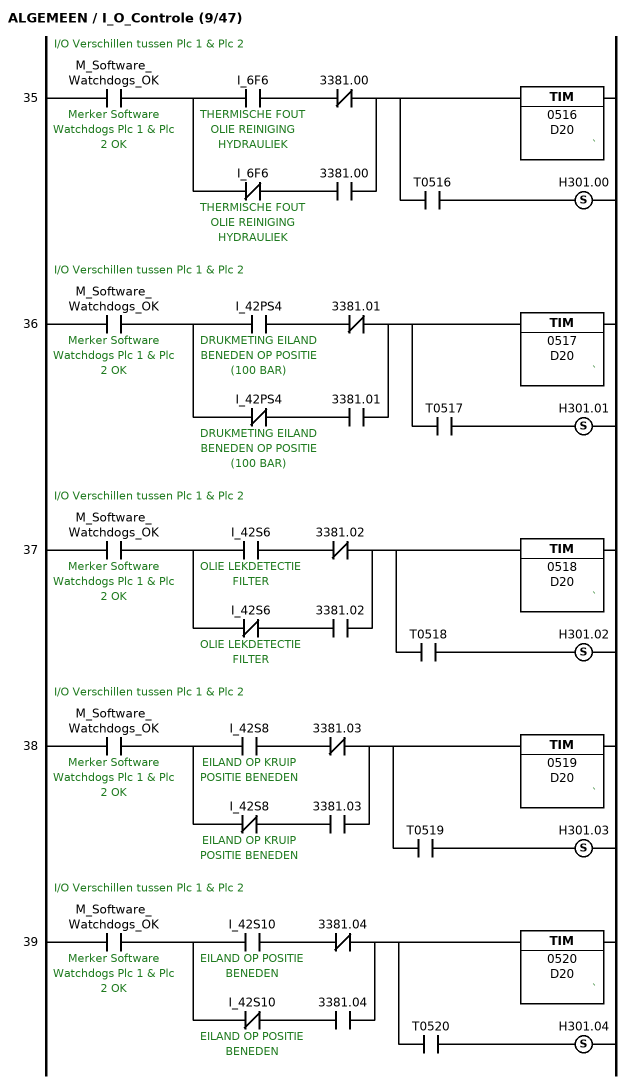
; [picture p24: ALGEMEEN / I_O_Controle, rungs 35-39]
; rung 35: I/O Verschillen tussen Plc 1 & Plc 2
LD M_Software_Watchdogs_OK  ; Merker Software Watchdogs Plc 1 & Plc 2 OK
LD I_6F6  ; THERMISCHE FOUT OLIE REINIGING HYDRAULIEK
ANDNOT 3381.00
LDNOT I_6F6  ; THERMISCHE FOUT OLIE REINIGING HYDRAULIEK
AND 3381.00
ORLD
ANDLD
TIM 0516 D20  ; `
AND T0516
SET H301.00
; rung 36: I/O Verschillen tussen Plc 1 & Plc 2
LD M_Software_Watchdogs_OK  ; Merker Software Watchdogs Plc 1 & Plc 2 OK
LD I_42PS4  ; DRUKMETING EILAND BENEDEN OP POSITIE (100 BAR)
ANDNOT 3381.01
LDNOT I_42PS4  ; DRUKMETING EILAND BENEDEN OP POSITIE (100 BAR)
AND 3381.01
ORLD
ANDLD
TIM 0517 D20  ; `
AND T0517
SET H301.01
; rung 37: I/O Verschillen tussen Plc 1 & Plc 2
LD M_Software_Watchdogs_OK  ; Merker Software Watchdogs Plc 1 & Plc 2 OK
LD I_42S6  ; OLIE LEKDETECTIE FILTER
ANDNOT 3381.02
LDNOT I_42S6  ; OLIE LEKDETECTIE FILTER
AND 3381.02
ORLD
ANDLD
TIM 0518 D20  ; `
AND T0518
SET H301.02
; rung 38: I/O Verschillen tussen Plc 1 & Plc 2
LD M_Software_Watchdogs_OK  ; Merker Software Watchdogs Plc 1 & Plc 2 OK
LD I_42S8  ; EILAND OP KRUIP POSITIE BENEDEN
ANDNOT 3381.03
LDNOT I_42S8  ; EILAND OP KRUIP POSITIE BENEDEN
AND 3381.03
ORLD
ANDLD
TIM 0519 D20  ; `
AND T0519
SET H301.03
; rung 39: I/O Verschillen tussen Plc 1 & Plc 2
LD M_Software_Watchdogs_OK  ; Merker Software Watchdogs Plc 1 & Plc 2 OK
LD I_42S10  ; EILAND OP POSITIE BENEDEN
ANDNOT 3381.04
LDNOT I_42S10  ; EILAND OP POSITIE BENEDEN
AND 3381.04
ORLD
ANDLD
TIM 0520 D20  ; `
AND T0520
SET H301.04

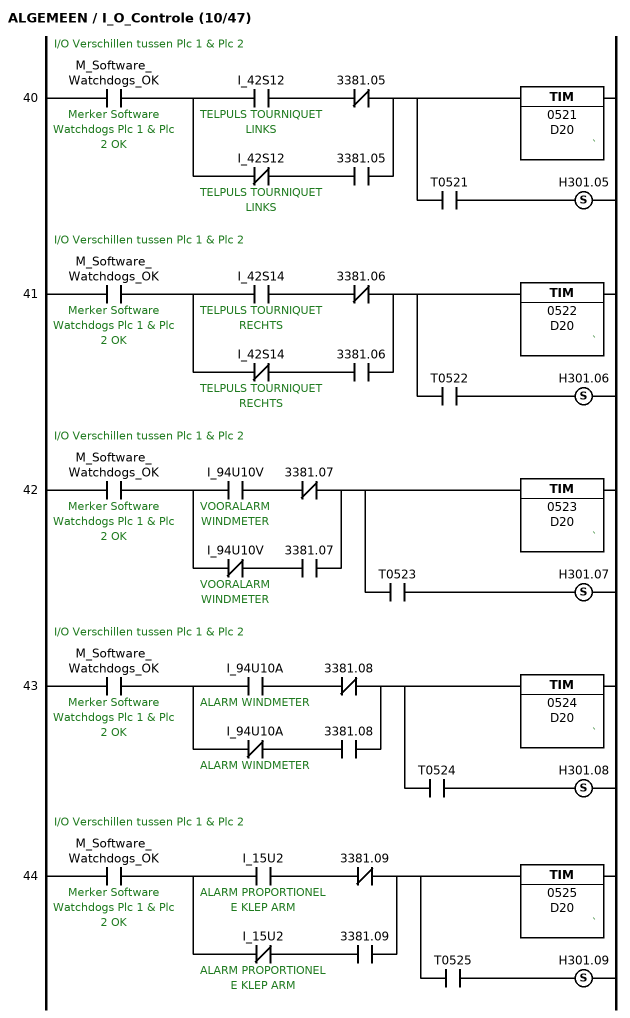
; rung 40: I/O Verschillen tussen Plc 1 & Plc 2
LD M_Software_Watchdogs_OK  ; Merker Software Watchdogs Plc 1 & Plc 2 OK
LD I_42S12  ; TELPULS TOURNIQUET LINKS
ANDNOT 3381.05
LDNOT I_42S12  ; TELPULS TOURNIQUET LINKS
AND 3381.05
ORLD
ANDLD
TIM 0521 D20  ; `
AND T0521
SET H301.05
; rung 41: I/O Verschillen tussen Plc 1 & Plc 2
LD M_Software_Watchdogs_OK  ; Merker Software Watchdogs Plc 1 & Plc 2 OK
LD I_42S14  ; TELPULS TOURNIQUET RECHTS
ANDNOT 3381.06
LDNOT I_42S14  ; TELPULS TOURNIQUET RECHTS
AND 3381.06
ORLD
ANDLD
TIM 0522 D20  ; `
AND T0522
SET H301.06
; rung 42: I/O Verschillen tussen Plc 1 & Plc 2
LD M_Software_Watchdogs_OK  ; Merker Software Watchdogs Plc 1 & Plc 2 OK
LD I_94U10V  ; VOORALARM WINDMETER
ANDNOT 3381.07
LDNOT I_94U10V  ; VOORALARM WINDMETER
AND 3381.07
ORLD
ANDLD
TIM 0523 D20  ; `
AND T0523
SET H301.07
; rung 43: I/O Verschillen tussen Plc 1 & Plc 2
LD M_Software_Watchdogs_OK  ; Merker Software Watchdogs Plc 1 & Plc 2 OK
LD I_94U10A  ; ALARM WINDMETER
ANDNOT 3381.08
LDNOT I_94U10A  ; ALARM WINDMETER
AND 3381.08
ORLD
ANDLD
TIM 0524 D20  ; `
AND T0524
SET H301.08
; rung 44: I/O Verschillen tussen Plc 1 & Plc 2
LD M_Software_Watchdogs_OK  ; Merker Software Watchdogs Plc 1 & Plc 2 OK
LD I_15U2  ; ALARM PROPORTIONELE KLEP ARM
ANDNOT 3381.09
LDNOT I_15U2  ; ALARM PROPORTIONELE KLEP ARM
AND 3381.09
ORLD
ANDLD
TIM 0525 D20  ; `
AND T0525
SET H301.09

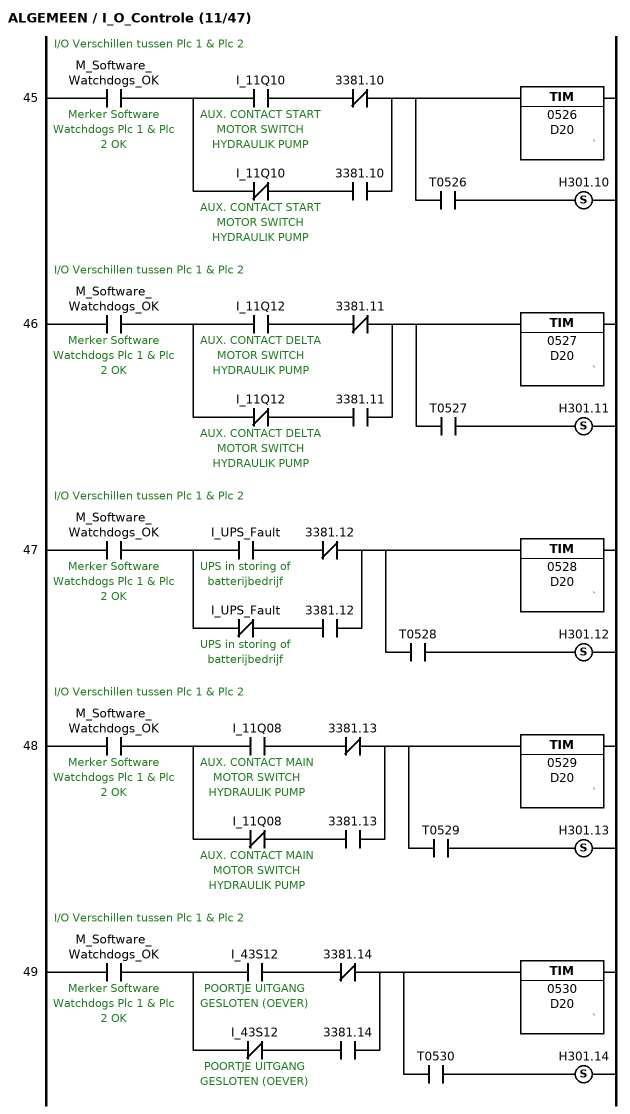
; rung 45: I/O Verschillen tussen Plc 1 & Plc 2
LD M_Software_Watchdogs_OK  ; Merker Software Watchdogs Plc 1 & Plc 2 OK
LD I_11Q10  ; AUX. CONTACT START MOTOR SWITCH HYDRAULIK PUMP
ANDNOT 3381.10
LDNOT I_11Q10  ; AUX. CONTACT START MOTOR SWITCH HYDRAULIK PUMP
AND 3381.10
ORLD
ANDLD
TIM 0526 D20  ; `
AND T0526
SET H301.10
; rung 46: I/O Verschillen tussen Plc 1 & Plc 2
LD M_Software_Watchdogs_OK  ; Merker Software Watchdogs Plc 1 & Plc 2 OK
LD I_11Q12  ; AUX. CONTACT DELTA MOTOR SWITCH HYDRAULIK PUMP
ANDNOT 3381.11
LDNOT I_11Q12  ; AUX. CONTACT DELTA MOTOR SWITCH HYDRAULIK PUMP
AND 3381.11
ORLD
ANDLD
TIM 0527 D20  ; `
AND T0527
SET H301.11
; rung 47: I/O Verschillen tussen Plc 1 & Plc 2
LD M_Software_Watchdogs_OK  ; Merker Software Watchdogs Plc 1 & Plc 2 OK
LD I_UPS_Fault  ; UPS in storing of batterijbedrijf
ANDNOT 3381.12
LDNOT I_UPS_Fault  ; UPS in storing of batterijbedrijf
AND 3381.12
ORLD
ANDLD
TIM 0528 D20  ; `
AND T0528
SET H301.12
; rung 48: I/O Verschillen tussen Plc 1 & Plc 2
LD M_Software_Watchdogs_OK  ; Merker Software Watchdogs Plc 1 & Plc 2 OK
LD I_11Q08  ; AUX. CONTACT MAIN MOTOR SWITCH HYDRAULIK PUMP
ANDNOT 3381.13
LDNOT I_11Q08  ; AUX. CONTACT MAIN MOTOR SWITCH HYDRAULIK PUMP
AND 3381.13
ORLD
ANDLD
TIM 0529 D20  ; `
AND T0529
SET H301.13
; rung 49: I/O Verschillen tussen Plc 1 & Plc 2
LD M_Software_Watchdogs_OK  ; Merker Software Watchdogs Plc 1 & Plc 2 OK
LD I_43S12  ; POORTJE UITGANG GESLOTEN (OEVER)
ANDNOT 3381.14
LDNOT I_43S12  ; POORTJE UITGANG GESLOTEN (OEVER)
AND 3381.14
ORLD
ANDLD
TIM 0530 D20  ; `
AND T0530
SET H301.14

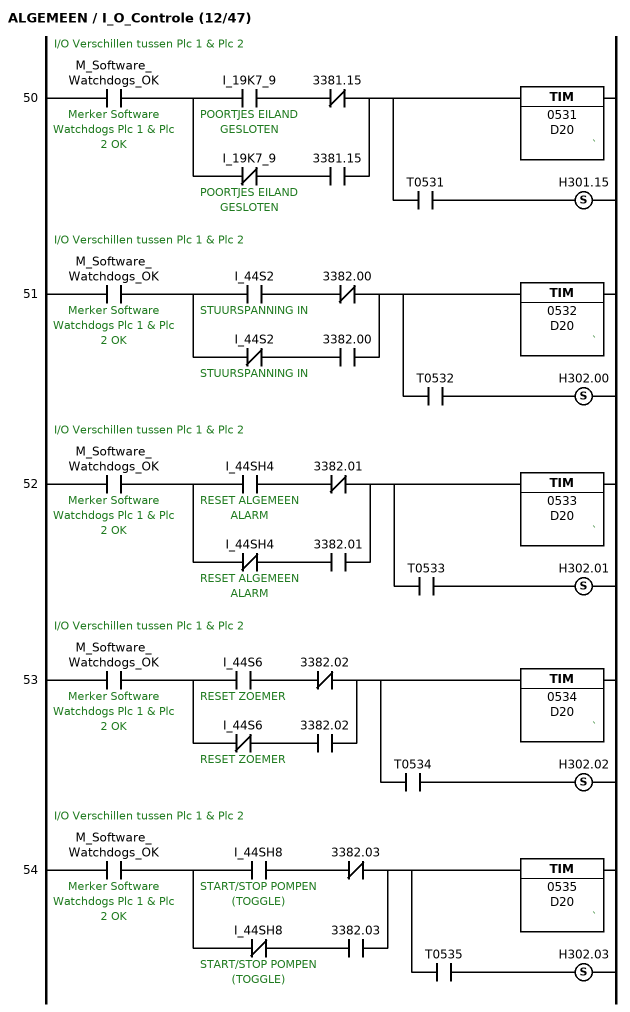
; rung 50: I/O Verschillen tussen Plc 1 & Plc 2
LD M_Software_Watchdogs_OK  ; Merker Software Watchdogs Plc 1 & Plc 2 OK
LD I_19K7_9  ; POORTJES EILAND GESLOTEN
ANDNOT 3381.15
LDNOT I_19K7_9  ; POORTJES EILAND GESLOTEN
AND 3381.15
ORLD
ANDLD
TIM 0531 D20  ; `
AND T0531
SET H301.15
; rung 51: I/O Verschillen tussen Plc 1 & Plc 2
LD M_Software_Watchdogs_OK  ; Merker Software Watchdogs Plc 1 & Plc 2 OK
LD I_44S2  ; STUURSPANNING IN
ANDNOT 3382.00
LDNOT I_44S2  ; STUURSPANNING IN
AND 3382.00
ORLD
ANDLD
TIM 0532 D20  ; `
AND T0532
SET H302.00
; rung 52: I/O Verschillen tussen Plc 1 & Plc 2
LD M_Software_Watchdogs_OK  ; Merker Software Watchdogs Plc 1 & Plc 2 OK
LD I_44SH4  ; RESET ALGEMEEN ALARM
ANDNOT 3382.01
LDNOT I_44SH4  ; RESET ALGEMEEN ALARM
AND 3382.01
ORLD
ANDLD
TIM 0533 D20  ; `
AND T0533
SET H302.01
; rung 53: I/O Verschillen tussen Plc 1 & Plc 2
LD M_Software_Watchdogs_OK  ; Merker Software Watchdogs Plc 1 & Plc 2 OK
LD I_44S6  ; RESET ZOEMER
ANDNOT 3382.02
LDNOT I_44S6  ; RESET ZOEMER
AND 3382.02
ORLD
ANDLD
TIM 0534 D20  ; `
AND T0534
SET H302.02
; rung 54: I/O Verschillen tussen Plc 1 & Plc 2
LD M_Software_Watchdogs_OK  ; Merker Software Watchdogs Plc 1 & Plc 2 OK
LD I_44SH8  ; START/STOP POMPEN (TOGGLE)
ANDNOT 3382.03
LDNOT I_44SH8  ; START/STOP POMPEN (TOGGLE)
AND 3382.03
ORLD
ANDLD
TIM 0535 D20  ; `
AND T0535
SET H302.03

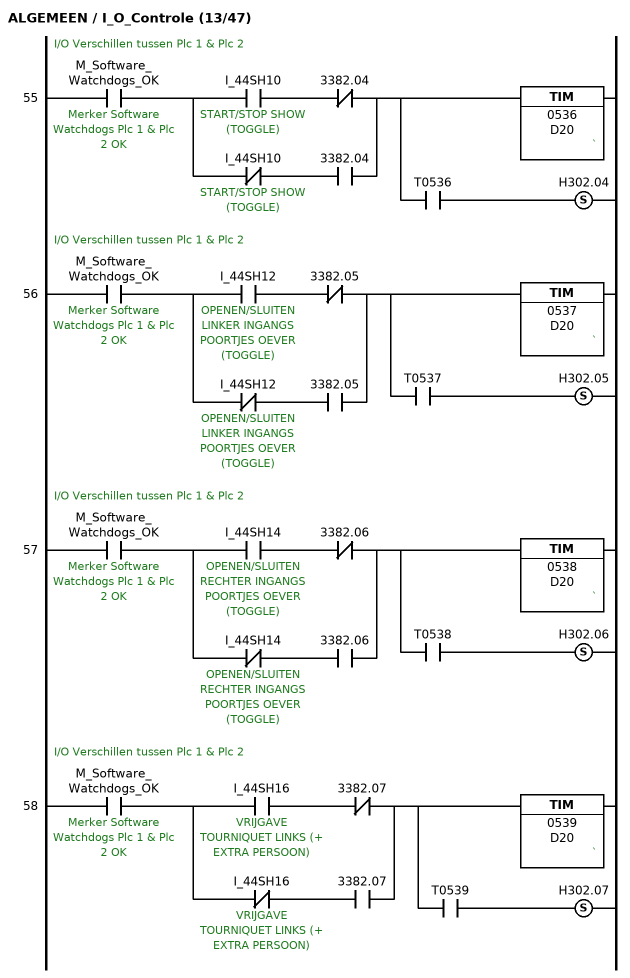
; rung 55: I/O Verschillen tussen Plc 1 & Plc 2
LD M_Software_Watchdogs_OK  ; Merker Software Watchdogs Plc 1 & Plc 2 OK
LD I_44SH10  ; START/STOP SHOW (TOGGLE)
ANDNOT 3382.04
LDNOT I_44SH10  ; START/STOP SHOW (TOGGLE)
AND 3382.04
ORLD
ANDLD
TIM 0536 D20  ; `
AND T0536
SET H302.04
; rung 56: I/O Verschillen tussen Plc 1 & Plc 2
LD M_Software_Watchdogs_OK  ; Merker Software Watchdogs Plc 1 & Plc 2 OK
LD I_44SH12  ; OPENEN/SLUITEN LINKER INGANGS POORTJES OEVER  (TOGGLE)
ANDNOT 3382.05
LDNOT I_44SH12  ; OPENEN/SLUITEN LINKER INGANGS POORTJES OEVER  (TOGGLE)
AND 3382.05
ORLD
ANDLD
TIM 0537 D20  ; `
AND T0537
SET H302.05
; rung 57: I/O Verschillen tussen Plc 1 & Plc 2
LD M_Software_Watchdogs_OK  ; Merker Software Watchdogs Plc 1 & Plc 2 OK
LD I_44SH14  ; OPENEN/SLUITEN RECHTER INGANGS POORTJES OEVER  (TOGGLE)
ANDNOT 3382.06
LDNOT I_44SH14  ; OPENEN/SLUITEN RECHTER INGANGS POORTJES OEVER  (TOGGLE)
AND 3382.06
ORLD
ANDLD
TIM 0538 D20  ; `
AND T0538
SET H302.06
; rung 58: I/O Verschillen tussen Plc 1 & Plc 2
LD M_Software_Watchdogs_OK  ; Merker Software Watchdogs Plc 1 & Plc 2 OK
LD I_44SH16  ; VRIJGAVE TOURNIQUET LINKS (+ EXTRA PERSOON)
ANDNOT 3382.07
LDNOT I_44SH16  ; VRIJGAVE TOURNIQUET LINKS (+ EXTRA PERSOON)
AND 3382.07
ORLD
ANDLD
TIM 0539 D20  ; `
AND T0539
SET H302.07

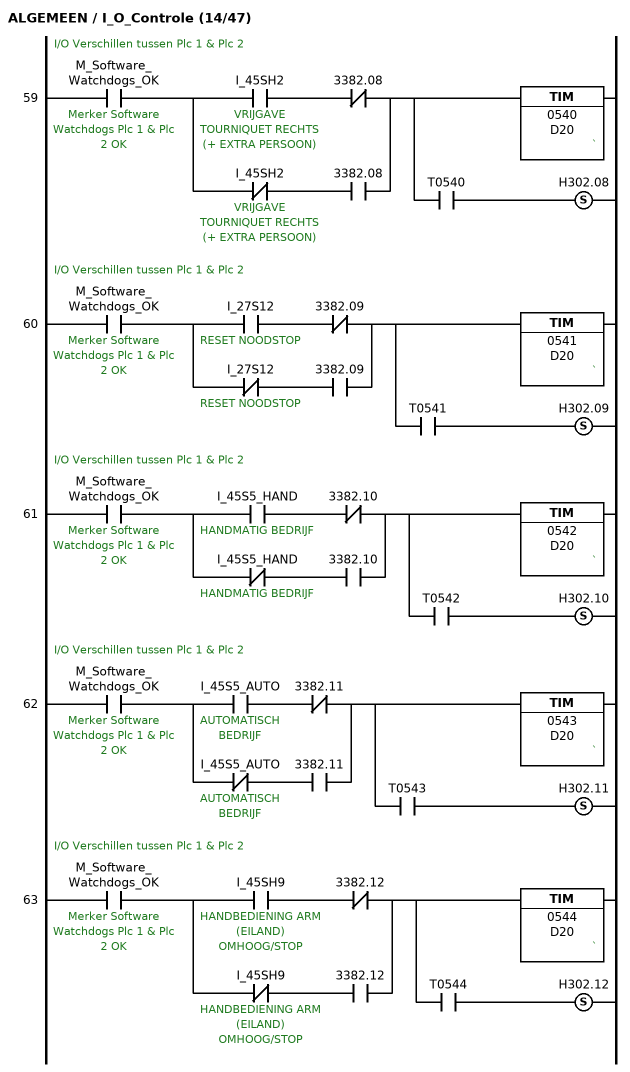
; rung 59: I/O Verschillen tussen Plc 1 & Plc 2
LD M_Software_Watchdogs_OK  ; Merker Software Watchdogs Plc 1 & Plc 2 OK
LD I_45SH2  ; VRIJGAVE TOURNIQUET RECHTS (+ EXTRA PERSOON)
ANDNOT 3382.08
LDNOT I_45SH2  ; VRIJGAVE TOURNIQUET RECHTS (+ EXTRA PERSOON)
AND 3382.08
ORLD
ANDLD
TIM 0540 D20  ; `
AND T0540
SET H302.08
; rung 60: I/O Verschillen tussen Plc 1 & Plc 2
LD M_Software_Watchdogs_OK  ; Merker Software Watchdogs Plc 1 & Plc 2 OK
LD I_27S12  ; RESET NOODSTOP
ANDNOT 3382.09
LDNOT I_27S12  ; RESET NOODSTOP
AND 3382.09
ORLD
ANDLD
TIM 0541 D20  ; `
AND T0541
SET H302.09
; rung 61: I/O Verschillen tussen Plc 1 & Plc 2
LD M_Software_Watchdogs_OK  ; Merker Software Watchdogs Plc 1 & Plc 2 OK
LD I_45S5_HAND  ; HANDMATIG BEDRIJF
ANDNOT 3382.10
LDNOT I_45S5_HAND  ; HANDMATIG BEDRIJF
AND 3382.10
ORLD
ANDLD
TIM 0542 D20  ; `
AND T0542
SET H302.10
; rung 62: I/O Verschillen tussen Plc 1 & Plc 2
LD M_Software_Watchdogs_OK  ; Merker Software Watchdogs Plc 1 & Plc 2 OK
LD I_45S5_AUTO  ; AUTOMATISCH BEDRIJF
ANDNOT 3382.11
LDNOT I_45S5_AUTO  ; AUTOMATISCH BEDRIJF
AND 3382.11
ORLD
ANDLD
TIM 0543 D20  ; `
AND T0543
SET H302.11
; rung 63: I/O Verschillen tussen Plc 1 & Plc 2
LD M_Software_Watchdogs_OK  ; Merker Software Watchdogs Plc 1 & Plc 2 OK
LD I_45SH9  ; HANDBEDIENING ARM (EILAND) OMHOOG/STOP
ANDNOT 3382.12
LDNOT I_45SH9  ; HANDBEDIENING ARM (EILAND) OMHOOG/STOP
AND 3382.12
ORLD
ANDLD
TIM 0544 D20  ; `
AND T0544
SET H302.12

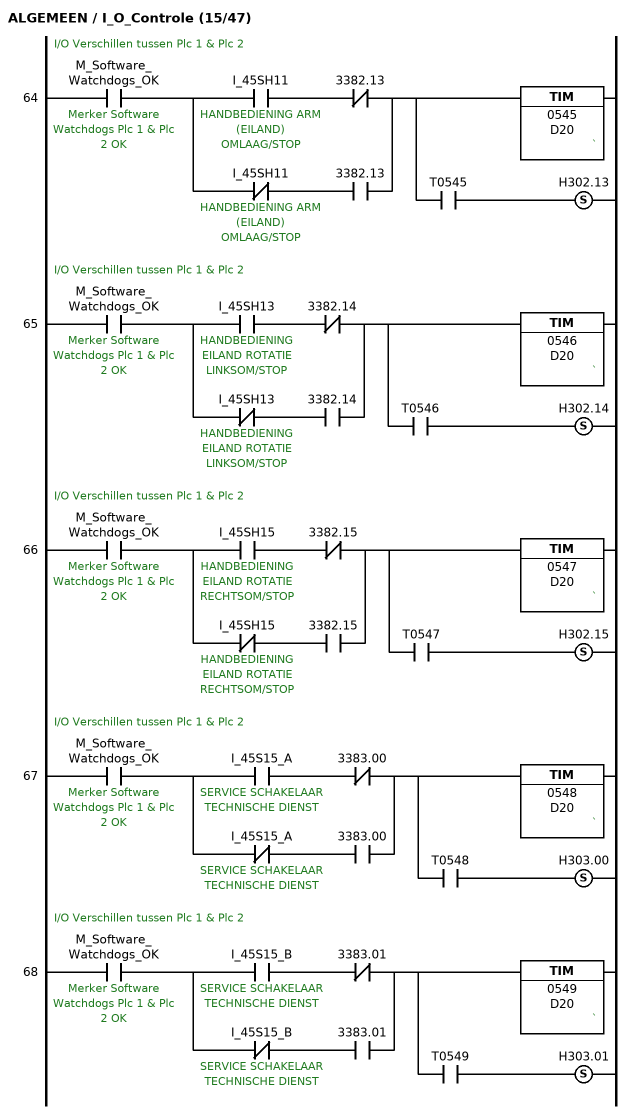
; rung 64: I/O Verschillen tussen Plc 1 & Plc 2
LD M_Software_Watchdogs_OK  ; Merker Software Watchdogs Plc 1 & Plc 2 OK
LD I_45SH11  ; HANDBEDIENING ARM (EILAND) OMLAAG/STOP
ANDNOT 3382.13
LDNOT I_45SH11  ; HANDBEDIENING ARM (EILAND) OMLAAG/STOP
AND 3382.13
ORLD
ANDLD
TIM 0545 D20  ; `
AND T0545
SET H302.13
; rung 65: I/O Verschillen tussen Plc 1 & Plc 2
LD M_Software_Watchdogs_OK  ; Merker Software Watchdogs Plc 1 & Plc 2 OK
LD I_45SH13  ; HANDBEDIENING EILAND ROTATIE LINKSOM/STOP
ANDNOT 3382.14
LDNOT I_45SH13  ; HANDBEDIENING EILAND ROTATIE LINKSOM/STOP
AND 3382.14
ORLD
ANDLD
TIM 0546 D20  ; `
AND T0546
SET H302.14
; rung 66: I/O Verschillen tussen Plc 1 & Plc 2
LD M_Software_Watchdogs_OK  ; Merker Software Watchdogs Plc 1 & Plc 2 OK
LD I_45SH15  ; HANDBEDIENING EILAND ROTATIE RECHTSOM/STOP
ANDNOT 3382.15
LDNOT I_45SH15  ; HANDBEDIENING EILAND ROTATIE RECHTSOM/STOP
AND 3382.15
ORLD
ANDLD
TIM 0547 D20  ; `
AND T0547
SET H302.15
; rung 67: I/O Verschillen tussen Plc 1 & Plc 2
LD M_Software_Watchdogs_OK  ; Merker Software Watchdogs Plc 1 & Plc 2 OK
LD I_45S15_A  ; SERVICE SCHAKELAAR TECHNISCHE DIENST
ANDNOT 3383.00
LDNOT I_45S15_A  ; SERVICE SCHAKELAAR TECHNISCHE DIENST
AND 3383.00
ORLD
ANDLD
TIM 0548 D20  ; `
AND T0548
SET H303.00
; rung 68: I/O Verschillen tussen Plc 1 & Plc 2
LD M_Software_Watchdogs_OK  ; Merker Software Watchdogs Plc 1 & Plc 2 OK
LD I_45S15_B  ; SERVICE SCHAKELAAR TECHNISCHE DIENST
ANDNOT 3383.01
LDNOT I_45S15_B  ; SERVICE SCHAKELAAR TECHNISCHE DIENST
AND 3383.01
ORLD
ANDLD
TIM 0549 D20  ; `
AND T0549
SET H303.01

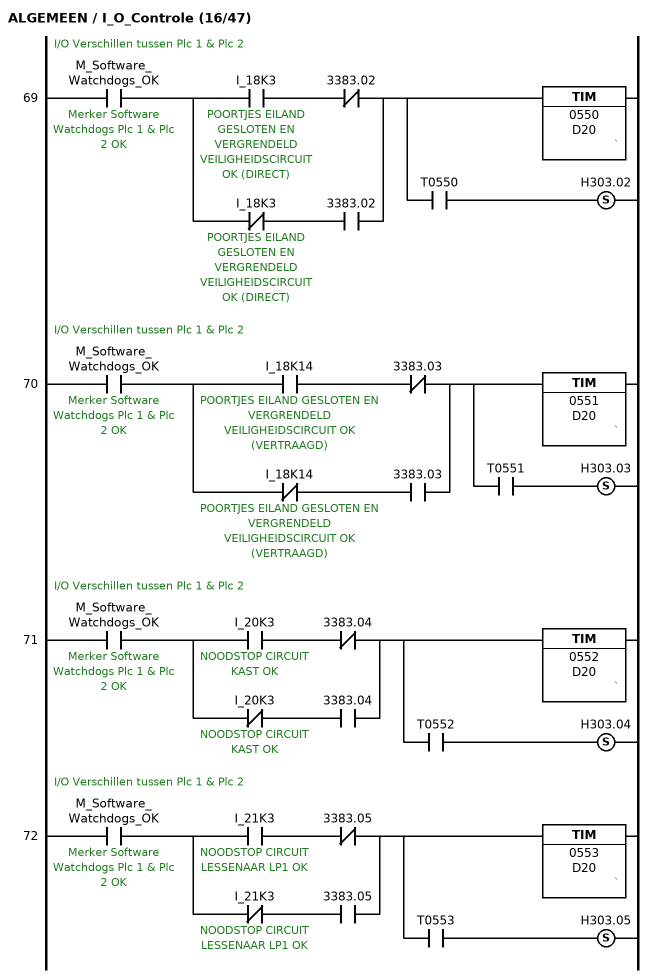
; rung 69: I/O Verschillen tussen Plc 1 & Plc 2
LD M_Software_Watchdogs_OK  ; Merker Software Watchdogs Plc 1 & Plc 2 OK
LD I_18K3  ; POORTJES EILAND GESLOTEN EN VERGRENDELD VEILIGHEIDSCIRCUIT OK (DIRECT)
ANDNOT 3383.02
LDNOT I_18K3  ; POORTJES EILAND GESLOTEN EN VERGRENDELD VEILIGHEIDSCIRCUIT OK (DIRECT)
AND 3383.02
ORLD
ANDLD
TIM 0550 D20  ; `
AND T0550
SET H303.02
; rung 70: I/O Verschillen tussen Plc 1 & Plc 2
LD M_Software_Watchdogs_OK  ; Merker Software Watchdogs Plc 1 & Plc 2 OK
LD I_18K14  ; POORTJES EILAND GESLOTEN EN VERGRENDELD VEILIGHEIDSCIRCUIT OK (VERTRAAGD)
ANDNOT 3383.03
LDNOT I_18K14  ; POORTJES EILAND GESLOTEN EN VERGRENDELD VEILIGHEIDSCIRCUIT OK (VERTRAAGD)
AND 3383.03
ORLD
ANDLD
TIM 0551 D20  ; `
AND T0551
SET H303.03
; rung 71: I/O Verschillen tussen Plc 1 & Plc 2
LD M_Software_Watchdogs_OK  ; Merker Software Watchdogs Plc 1 & Plc 2 OK
LD I_20K3  ; NOODSTOP CIRCUIT KAST OK
ANDNOT 3383.04
LDNOT I_20K3  ; NOODSTOP CIRCUIT KAST OK
AND 3383.04
ORLD
ANDLD
TIM 0552 D20  ; `
AND T0552
SET H303.04
; rung 72: I/O Verschillen tussen Plc 1 & Plc 2
LD M_Software_Watchdogs_OK  ; Merker Software Watchdogs Plc 1 & Plc 2 OK
LD I_21K3  ; NOODSTOP CIRCUIT LESSENAAR LP1 OK
ANDNOT 3383.05
LDNOT I_21K3  ; NOODSTOP CIRCUIT LESSENAAR LP1 OK
AND 3383.05
ORLD
ANDLD
TIM 0553 D20  ; `
AND T0553
SET H303.05

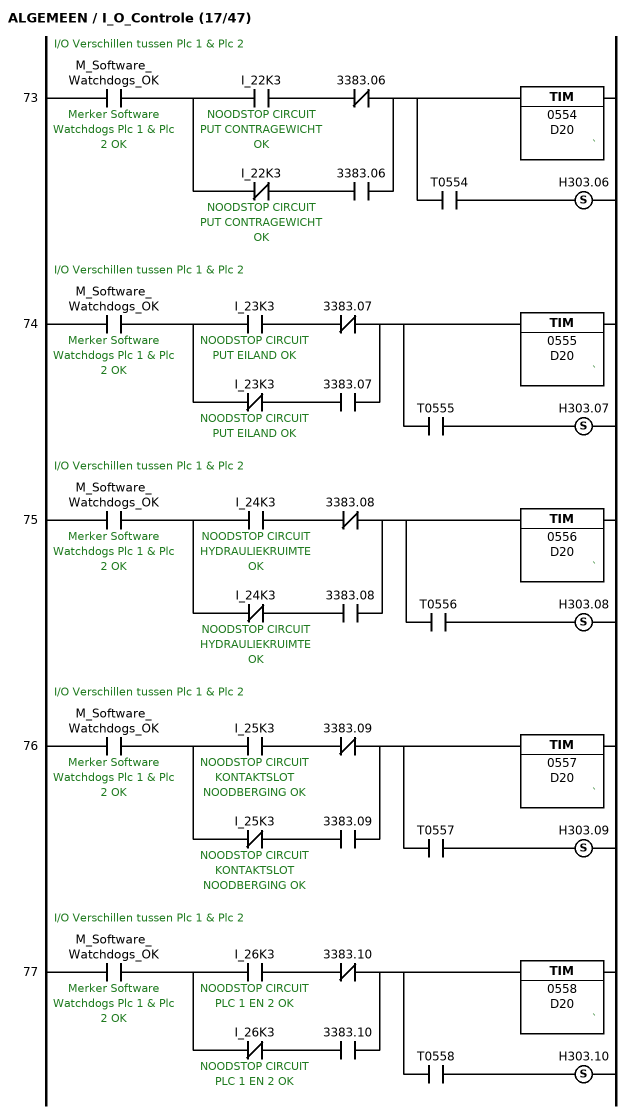
; rung 73: I/O Verschillen tussen Plc 1 & Plc 2
LD M_Software_Watchdogs_OK  ; Merker Software Watchdogs Plc 1 & Plc 2 OK
LD I_22K3  ; NOODSTOP CIRCUIT PUT CONTRAGEWICHT OK
ANDNOT 3383.06
LDNOT I_22K3  ; NOODSTOP CIRCUIT PUT CONTRAGEWICHT OK
AND 3383.06
ORLD
ANDLD
TIM 0554 D20  ; `
AND T0554
SET H303.06
; rung 74: I/O Verschillen tussen Plc 1 & Plc 2
LD M_Software_Watchdogs_OK  ; Merker Software Watchdogs Plc 1 & Plc 2 OK
LD I_23K3  ; NOODSTOP CIRCUIT PUT EILAND OK
ANDNOT 3383.07
LDNOT I_23K3  ; NOODSTOP CIRCUIT PUT EILAND OK
AND 3383.07
ORLD
ANDLD
TIM 0555 D20  ; `
AND T0555
SET H303.07
; rung 75: I/O Verschillen tussen Plc 1 & Plc 2
LD M_Software_Watchdogs_OK  ; Merker Software Watchdogs Plc 1 & Plc 2 OK
LD I_24K3  ; NOODSTOP CIRCUIT HYDRAULIEKRUIMTE OK
ANDNOT 3383.08
LDNOT I_24K3  ; NOODSTOP CIRCUIT HYDRAULIEKRUIMTE OK
AND 3383.08
ORLD
ANDLD
TIM 0556 D20  ; `
AND T0556
SET H303.08
; rung 76: I/O Verschillen tussen Plc 1 & Plc 2
LD M_Software_Watchdogs_OK  ; Merker Software Watchdogs Plc 1 & Plc 2 OK
LD I_25K3  ; NOODSTOP CIRCUIT KONTAKTSLOT NOODBERGING OK
ANDNOT 3383.09
LDNOT I_25K3  ; NOODSTOP CIRCUIT KONTAKTSLOT NOODBERGING OK
AND 3383.09
ORLD
ANDLD
TIM 0557 D20  ; `
AND T0557
SET H303.09
; rung 77: I/O Verschillen tussen Plc 1 & Plc 2
LD M_Software_Watchdogs_OK  ; Merker Software Watchdogs Plc 1 & Plc 2 OK
LD I_26K3  ; NOODSTOP CIRCUIT PLC 1 EN 2 OK
ANDNOT 3383.10
LDNOT I_26K3  ; NOODSTOP CIRCUIT PLC 1 EN 2 OK
AND 3383.10
ORLD
ANDLD
TIM 0558 D20  ; `
AND T0558
SET H303.10

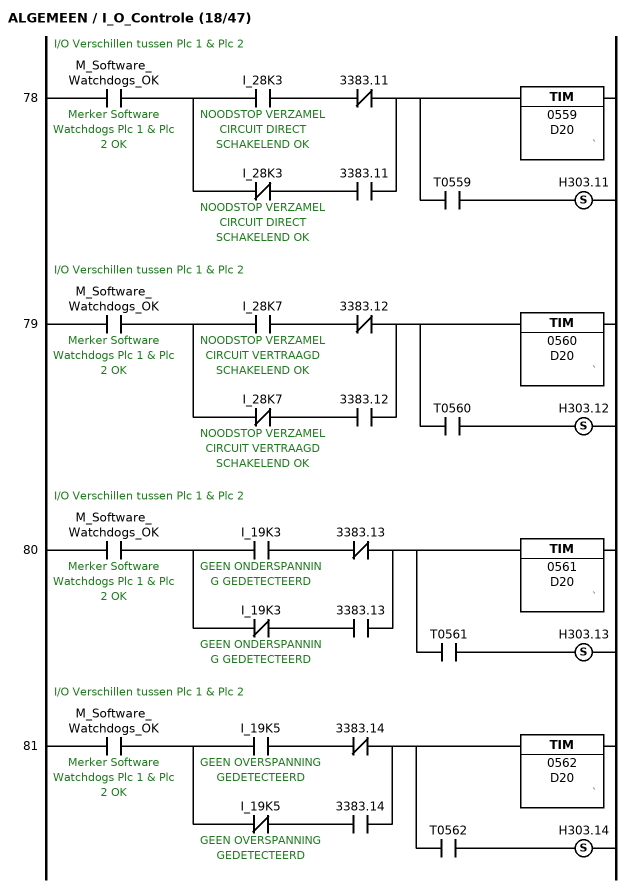
; rung 78: I/O Verschillen tussen Plc 1 & Plc 2
LD M_Software_Watchdogs_OK  ; Merker Software Watchdogs Plc 1 & Plc 2 OK
LD I_28K3  ; NOODSTOP VERZAMEL CIRCUIT DIRECT SCHAKELEND OK
ANDNOT 3383.11
LDNOT I_28K3  ; NOODSTOP VERZAMEL CIRCUIT DIRECT SCHAKELEND OK
AND 3383.11
ORLD
ANDLD
TIM 0559 D20  ; `
AND T0559
SET H303.11
; rung 79: I/O Verschillen tussen Plc 1 & Plc 2
LD M_Software_Watchdogs_OK  ; Merker Software Watchdogs Plc 1 & Plc 2 OK
LD I_28K7  ; NOODSTOP VERZAMEL CIRCUIT VERTRAAGD SCHAKELEND OK
ANDNOT 3383.12
LDNOT I_28K7  ; NOODSTOP VERZAMEL CIRCUIT VERTRAAGD SCHAKELEND OK
AND 3383.12
ORLD
ANDLD
TIM 0560 D20  ; `
AND T0560
SET H303.12
; rung 80: I/O Verschillen tussen Plc 1 & Plc 2
LD M_Software_Watchdogs_OK  ; Merker Software Watchdogs Plc 1 & Plc 2 OK
LD I_19K3  ; GEEN ONDERSPANNING GEDETECTEERD
ANDNOT 3383.13
LDNOT I_19K3  ; GEEN ONDERSPANNING GEDETECTEERD
AND 3383.13
ORLD
ANDLD
TIM 0561 D20  ; `
AND T0561
SET H303.13
; rung 81: I/O Verschillen tussen Plc 1 & Plc 2
LD M_Software_Watchdogs_OK  ; Merker Software Watchdogs Plc 1 & Plc 2 OK
LD I_19K5  ; GEEN OVERSPANNING GEDETECTEERD
ANDNOT 3383.14
LDNOT I_19K5  ; GEEN OVERSPANNING GEDETECTEERD
AND 3383.14
ORLD
ANDLD
TIM 0562 D20  ; `
AND T0562
SET H303.14

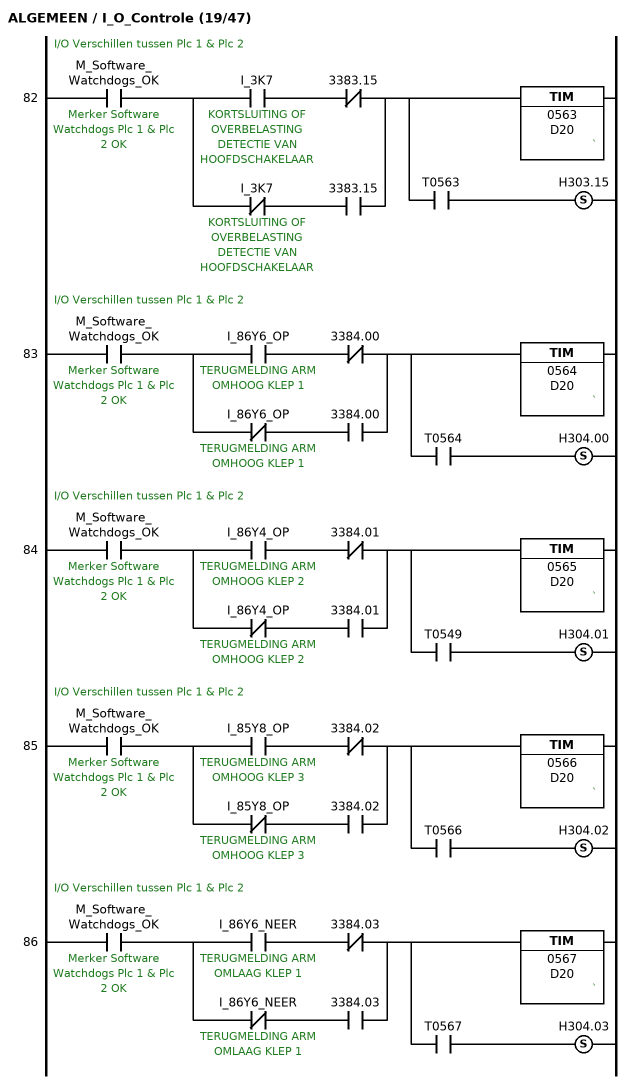
; rung 82: I/O Verschillen tussen Plc 1 & Plc 2
LD M_Software_Watchdogs_OK  ; Merker Software Watchdogs Plc 1 & Plc 2 OK
LD I_3K7  ; KORTSLUITING OF OVERBELASTING DETECTIE VAN HOOFDSCHAKELAAR
ANDNOT 3383.15
LDNOT I_3K7  ; KORTSLUITING OF OVERBELASTING DETECTIE VAN HOOFDSCHAKELAAR
AND 3383.15
ORLD
ANDLD
TIM 0563 D20  ; `
AND T0563
SET H303.15
; rung 83: I/O Verschillen tussen Plc 1 & Plc 2
LD M_Software_Watchdogs_OK  ; Merker Software Watchdogs Plc 1 & Plc 2 OK
LD I_86Y6_OP  ; TERUGMELDING ARM OMHOOG KLEP 1
ANDNOT 3384.00
LDNOT I_86Y6_OP  ; TERUGMELDING ARM OMHOOG KLEP 1
AND 3384.00
ORLD
ANDLD
TIM 0564 D20  ; `
AND T0564
SET H304.00
; rung 84: I/O Verschillen tussen Plc 1 & Plc 2
LD M_Software_Watchdogs_OK  ; Merker Software Watchdogs Plc 1 & Plc 2 OK
LD I_86Y4_OP  ; TERUGMELDING ARM OMHOOG KLEP 2
ANDNOT 3384.01
LDNOT I_86Y4_OP  ; TERUGMELDING ARM OMHOOG KLEP 2
AND 3384.01
ORLD
ANDLD
TIM 0565 D20  ; `
AND T0549
SET H304.01
; rung 85: I/O Verschillen tussen Plc 1 & Plc 2
LD M_Software_Watchdogs_OK  ; Merker Software Watchdogs Plc 1 & Plc 2 OK
LD I_85Y8_OP  ; TERUGMELDING ARM OMHOOG KLEP 3
ANDNOT 3384.02
LDNOT I_85Y8_OP  ; TERUGMELDING ARM OMHOOG KLEP 3
AND 3384.02
ORLD
ANDLD
TIM 0566 D20  ; `
AND T0566
SET H304.02
; rung 86: I/O Verschillen tussen Plc 1 & Plc 2
LD M_Software_Watchdogs_OK  ; Merker Software Watchdogs Plc 1 & Plc 2 OK
LD I_86Y6_NEER  ; TERUGMELDING ARM OMLAAG KLEP 1
ANDNOT 3384.03
LDNOT I_86Y6_NEER  ; TERUGMELDING ARM OMLAAG KLEP 1
AND 3384.03
ORLD
ANDLD
TIM 0567 D20  ; `
AND T0567
SET H304.03

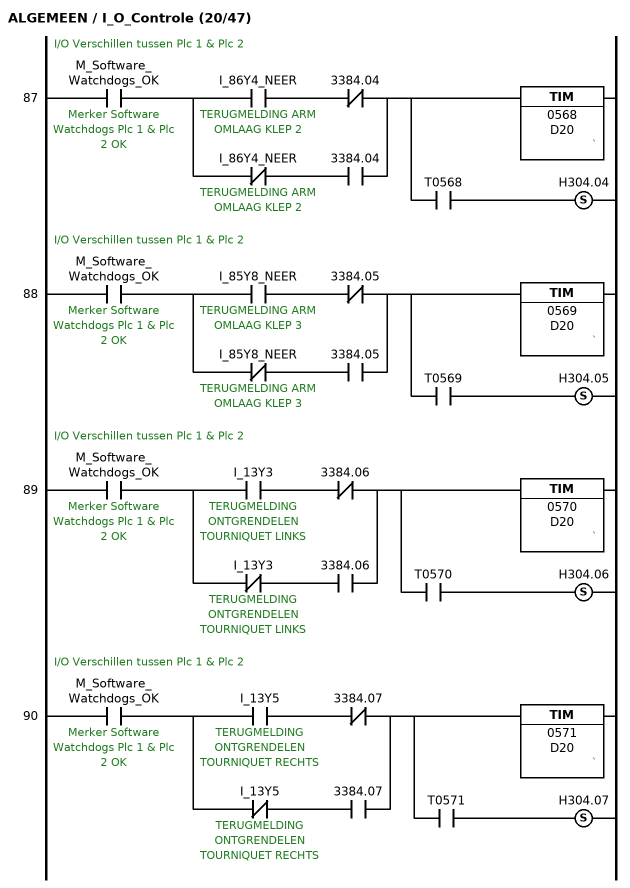
; rung 87: I/O Verschillen tussen Plc 1 & Plc 2
LD M_Software_Watchdogs_OK  ; Merker Software Watchdogs Plc 1 & Plc 2 OK
LD I_86Y4_NEER  ; TERUGMELDING ARM OMLAAG KLEP 2
ANDNOT 3384.04
LDNOT I_86Y4_NEER  ; TERUGMELDING ARM OMLAAG KLEP 2
AND 3384.04
ORLD
ANDLD
TIM 0568 D20  ; `
AND T0568
SET H304.04
; rung 88: I/O Verschillen tussen Plc 1 & Plc 2
LD M_Software_Watchdogs_OK  ; Merker Software Watchdogs Plc 1 & Plc 2 OK
LD I_85Y8_NEER  ; TERUGMELDING ARM OMLAAG KLEP 3
ANDNOT 3384.05
LDNOT I_85Y8_NEER  ; TERUGMELDING ARM OMLAAG KLEP 3
AND 3384.05
ORLD
ANDLD
TIM 0569 D20  ; `
AND T0569
SET H304.05
; rung 89: I/O Verschillen tussen Plc 1 & Plc 2
LD M_Software_Watchdogs_OK  ; Merker Software Watchdogs Plc 1 & Plc 2 OK
LD I_13Y3  ; TERUGMELDING ONTGRENDELEN TOURNIQUET LINKS
ANDNOT 3384.06
LDNOT I_13Y3  ; TERUGMELDING ONTGRENDELEN TOURNIQUET LINKS
AND 3384.06
ORLD
ANDLD
TIM 0570 D20  ; `
AND T0570
SET H304.06
; rung 90: I/O Verschillen tussen Plc 1 & Plc 2
LD M_Software_Watchdogs_OK  ; Merker Software Watchdogs Plc 1 & Plc 2 OK
LD I_13Y5  ; TERUGMELDING ONTGRENDELEN TOURNIQUET RECHTS
ANDNOT 3384.07
LDNOT I_13Y5  ; TERUGMELDING ONTGRENDELEN TOURNIQUET RECHTS
AND 3384.07
ORLD
ANDLD
TIM 0571 D20  ; `
AND T0571
SET H304.07

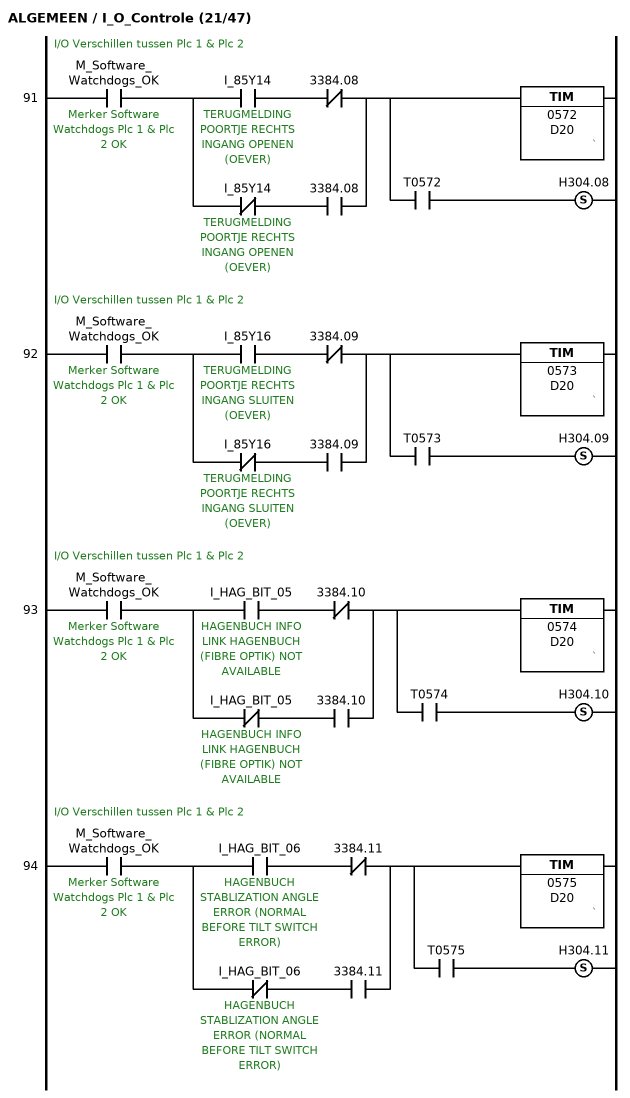
; rung 91: I/O Verschillen tussen Plc 1 & Plc 2
LD M_Software_Watchdogs_OK  ; Merker Software Watchdogs Plc 1 & Plc 2 OK
LD I_85Y14  ; TERUGMELDING POORTJE RECHTS INGANG OPENEN (OEVER)
ANDNOT 3384.08
LDNOT I_85Y14  ; TERUGMELDING POORTJE RECHTS INGANG OPENEN (OEVER)
AND 3384.08
ORLD
ANDLD
TIM 0572 D20  ; `
AND T0572
SET H304.08
; rung 92: I/O Verschillen tussen Plc 1 & Plc 2
LD M_Software_Watchdogs_OK  ; Merker Software Watchdogs Plc 1 & Plc 2 OK
LD I_85Y16  ; TERUGMELDING POORTJE RECHTS INGANG SLUITEN (OEVER)
ANDNOT 3384.09
LDNOT I_85Y16  ; TERUGMELDING POORTJE RECHTS INGANG SLUITEN (OEVER)
AND 3384.09
ORLD
ANDLD
TIM 0573 D20  ; `
AND T0573
SET H304.09
; rung 93: I/O Verschillen tussen Plc 1 & Plc 2
LD M_Software_Watchdogs_OK  ; Merker Software Watchdogs Plc 1 & Plc 2 OK
LD I_HAG_BIT_05  ; HAGENBUCH INFO LINK HAGENBUCH (FIBRE OPTIK) NOT AVAILABLE
ANDNOT 3384.10
LDNOT I_HAG_BIT_05  ; HAGENBUCH INFO LINK HAGENBUCH (FIBRE OPTIK) NOT AVAILABLE
AND 3384.10
ORLD
ANDLD
TIM 0574 D20  ; `
AND T0574
SET H304.10
; rung 94: I/O Verschillen tussen Plc 1 & Plc 2
LD M_Software_Watchdogs_OK  ; Merker Software Watchdogs Plc 1 & Plc 2 OK
LD I_HAG_BIT_06  ; HAGENBUCH STABLIZATION ANGLE ERROR (NORMAL BEFORE TILT SWITCH ERROR)
ANDNOT 3384.11
LDNOT I_HAG_BIT_06  ; HAGENBUCH STABLIZATION ANGLE ERROR (NORMAL BEFORE TILT SWITCH ERROR)
AND 3384.11
ORLD
ANDLD
TIM 0575 D20  ; `
AND T0575
SET H304.11

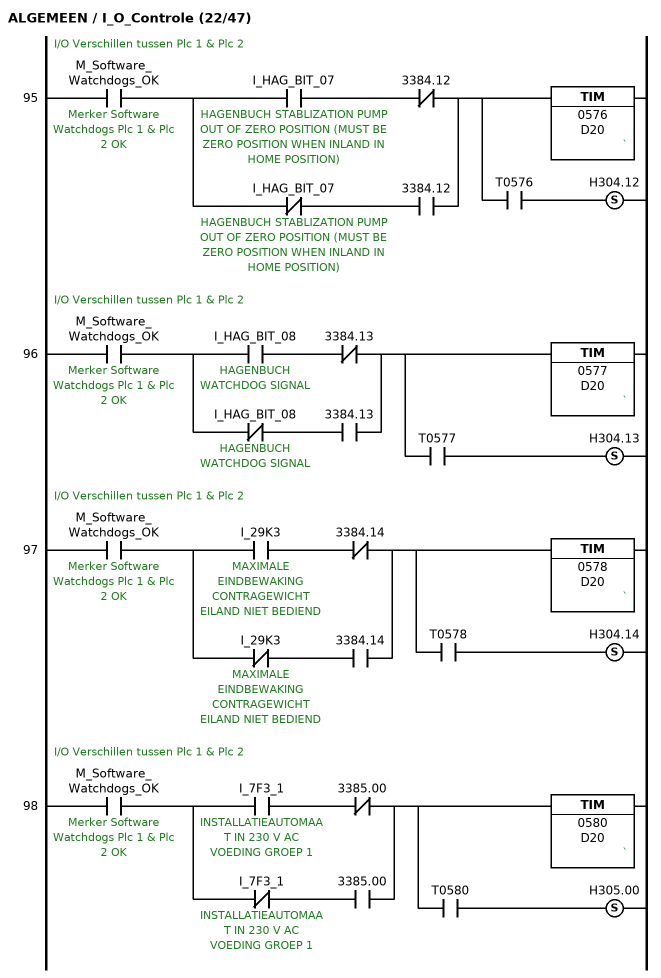
; rung 95: I/O Verschillen tussen Plc 1 & Plc 2
LD M_Software_Watchdogs_OK  ; Merker Software Watchdogs Plc 1 & Plc 2 OK
LD I_HAG_BIT_07  ; HAGENBUCH STABLIZATION PUMP OUT OF ZERO POSITION (MUST BE ZERO POSITION WHEN INLAND IN HOME POSITION)
ANDNOT 3384.12
LDNOT I_HAG_BIT_07  ; HAGENBUCH STABLIZATION PUMP OUT OF ZERO POSITION (MUST BE ZERO POSITION WHEN INLAND IN HOME POSITION)
AND 3384.12
ORLD
ANDLD
TIM 0576 D20  ; `
AND T0576
SET H304.12
; rung 96: I/O Verschillen tussen Plc 1 & Plc 2
LD M_Software_Watchdogs_OK  ; Merker Software Watchdogs Plc 1 & Plc 2 OK
LD I_HAG_BIT_08  ; HAGENBUCH WATCHDOG SIGNAL
ANDNOT 3384.13
LDNOT I_HAG_BIT_08  ; HAGENBUCH WATCHDOG SIGNAL
AND 3384.13
ORLD
ANDLD
TIM 0577 D20  ; `
AND T0577
SET H304.13
; rung 97: I/O Verschillen tussen Plc 1 & Plc 2
LD M_Software_Watchdogs_OK  ; Merker Software Watchdogs Plc 1 & Plc 2 OK
LD I_29K3  ; MAXIMALE EINDBEWAKING CONTRAGEWICHT EILAND NIET BEDIEND
ANDNOT 3384.14
LDNOT I_29K3  ; MAXIMALE EINDBEWAKING CONTRAGEWICHT EILAND NIET BEDIEND
AND 3384.14
ORLD
ANDLD
TIM 0578 D20  ; `
AND T0578
SET H304.14
; rung 98: I/O Verschillen tussen Plc 1 & Plc 2
LD M_Software_Watchdogs_OK  ; Merker Software Watchdogs Plc 1 & Plc 2 OK
LD I_7F3_1  ; INSTALLATIEAUTOMAAT IN 230 V AC VOEDING GROEP 1
ANDNOT 3385.00
LDNOT I_7F3_1  ; INSTALLATIEAUTOMAAT IN 230 V AC VOEDING GROEP 1
AND 3385.00
ORLD
ANDLD
TIM 0580 D20  ; `
AND T0580
SET H305.00

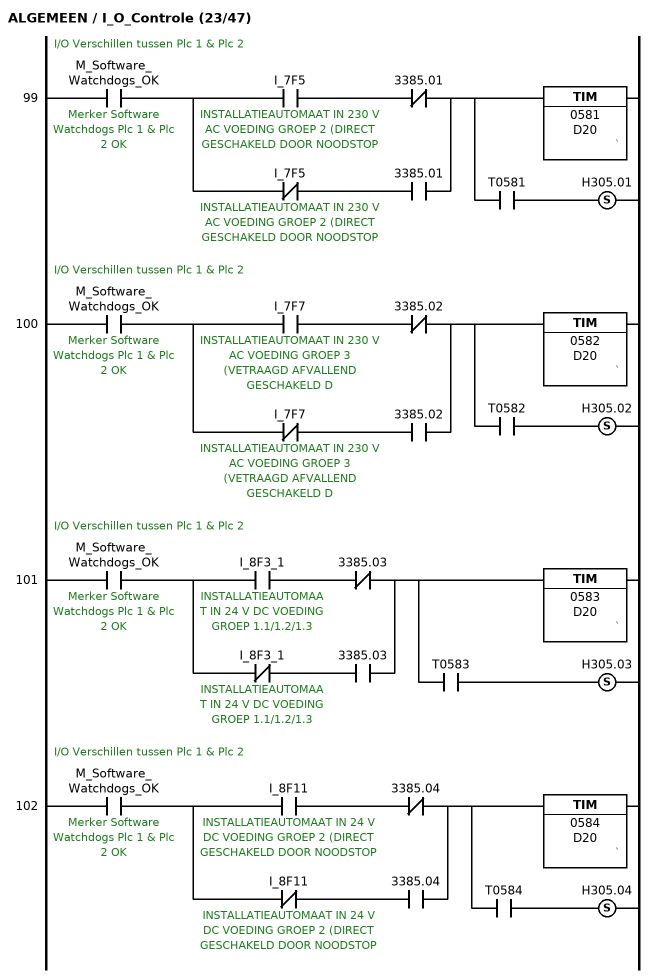
; rung 99: I/O Verschillen tussen Plc 1 & Plc 2
LD M_Software_Watchdogs_OK  ; Merker Software Watchdogs Plc 1 & Plc 2 OK
LD I_7F5  ; INSTALLATIEAUTOMAAT IN 230 V AC VOEDING GROEP 2 (DIRECT GESCHAKELD DOOR NOODSTOP
ANDNOT 3385.01
LDNOT I_7F5  ; INSTALLATIEAUTOMAAT IN 230 V AC VOEDING GROEP 2 (DIRECT GESCHAKELD DOOR NOODSTOP
AND 3385.01
ORLD
ANDLD
TIM 0581 D20  ; `
AND T0581
SET H305.01
; rung 100: I/O Verschillen tussen Plc 1 & Plc 2
LD M_Software_Watchdogs_OK  ; Merker Software Watchdogs Plc 1 & Plc 2 OK
LD I_7F7  ; INSTALLATIEAUTOMAAT IN 230 V AC VOEDING GROEP 3 (VETRAAGD AFVALLEND GESCHAKELD D
ANDNOT 3385.02
LDNOT I_7F7  ; INSTALLATIEAUTOMAAT IN 230 V AC VOEDING GROEP 3 (VETRAAGD AFVALLEND GESCHAKELD D
AND 3385.02
ORLD
ANDLD
TIM 0582 D20  ; `
AND T0582
SET H305.02
; rung 101: I/O Verschillen tussen Plc 1 & Plc 2
LD M_Software_Watchdogs_OK  ; Merker Software Watchdogs Plc 1 & Plc 2 OK
LD I_8F3_1  ; INSTALLATIEAUTOMAAT IN 24 V DC VOEDING GROEP 1.1/1.2/1.3
ANDNOT 3385.03
LDNOT I_8F3_1  ; INSTALLATIEAUTOMAAT IN 24 V DC VOEDING GROEP 1.1/1.2/1.3
AND 3385.03
ORLD
ANDLD
TIM 0583 D20  ; `
AND T0583
SET H305.03
; rung 102: I/O Verschillen tussen Plc 1 & Plc 2
LD M_Software_Watchdogs_OK  ; Merker Software Watchdogs Plc 1 & Plc 2 OK
LD I_8F11  ; INSTALLATIEAUTOMAAT IN 24 V DC VOEDING GROEP 2 (DIRECT GESCHAKELD DOOR NOODSTOP
ANDNOT 3385.04
LDNOT I_8F11  ; INSTALLATIEAUTOMAAT IN 24 V DC VOEDING GROEP 2 (DIRECT GESCHAKELD DOOR NOODSTOP
AND 3385.04
ORLD
ANDLD
TIM 0584 D20  ; `
AND T0584
SET H305.04

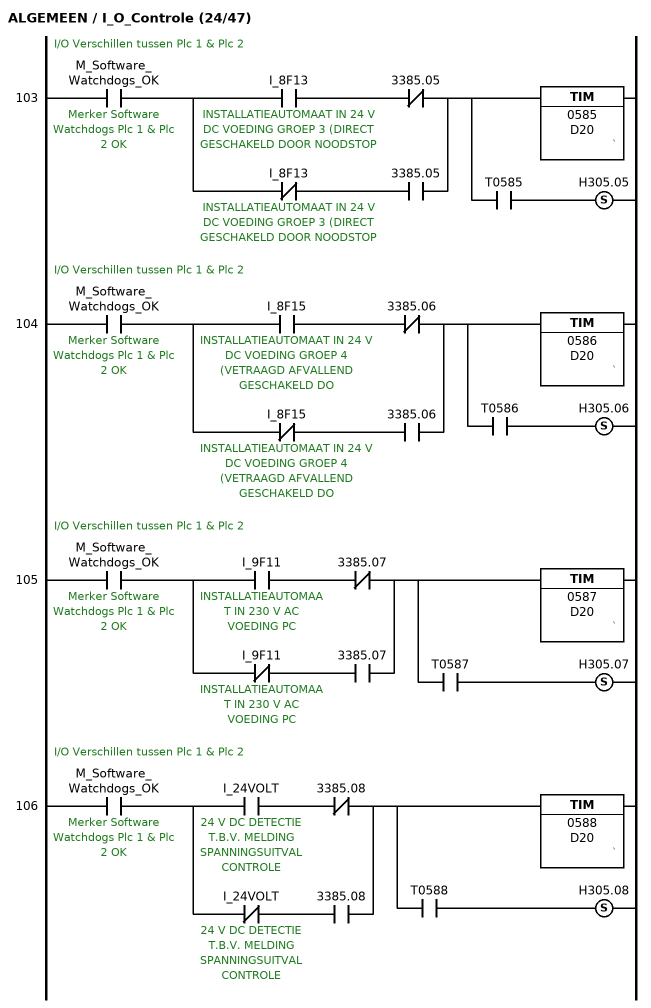
; rung 103: I/O Verschillen tussen Plc 1 & Plc 2
LD M_Software_Watchdogs_OK  ; Merker Software Watchdogs Plc 1 & Plc 2 OK
LD I_8F13  ; INSTALLATIEAUTOMAAT IN 24 V DC VOEDING GROEP 3 (DIRECT GESCHAKELD DOOR NOODSTOP
ANDNOT 3385.05
LDNOT I_8F13  ; INSTALLATIEAUTOMAAT IN 24 V DC VOEDING GROEP 3 (DIRECT GESCHAKELD DOOR NOODSTOP
AND 3385.05
ORLD
ANDLD
TIM 0585 D20  ; `
AND T0585
SET H305.05
; rung 104: I/O Verschillen tussen Plc 1 & Plc 2
LD M_Software_Watchdogs_OK  ; Merker Software Watchdogs Plc 1 & Plc 2 OK
LD I_8F15  ; INSTALLATIEAUTOMAAT IN 24 V DC VOEDING GROEP 4 (VETRAAGD AFVALLEND GESCHAKELD DO
ANDNOT 3385.06
LDNOT I_8F15  ; INSTALLATIEAUTOMAAT IN 24 V DC VOEDING GROEP 4 (VETRAAGD AFVALLEND GESCHAKELD DO
AND 3385.06
ORLD
ANDLD
TIM 0586 D20  ; `
AND T0586
SET H305.06
; rung 105: I/O Verschillen tussen Plc 1 & Plc 2
LD M_Software_Watchdogs_OK  ; Merker Software Watchdogs Plc 1 & Plc 2 OK
LD I_9F11  ; INSTALLATIEAUTOMAAT IN 230 V AC VOEDING PC
ANDNOT 3385.07
LDNOT I_9F11  ; INSTALLATIEAUTOMAAT IN 230 V AC VOEDING PC
AND 3385.07
ORLD
ANDLD
TIM 0587 D20  ; `
AND T0587
SET H305.07
; rung 106: I/O Verschillen tussen Plc 1 & Plc 2
LD M_Software_Watchdogs_OK  ; Merker Software Watchdogs Plc 1 & Plc 2 OK
LD I_24VOLT  ; 24 V DC DETECTIE T.B.V. MELDING SPANNINGSUITVAL CONTROLE
ANDNOT 3385.08
LDNOT I_24VOLT  ; 24 V DC DETECTIE T.B.V. MELDING SPANNINGSUITVAL CONTROLE
AND 3385.08
ORLD
ANDLD
TIM 0588 D20  ; `
AND T0588
SET H305.08

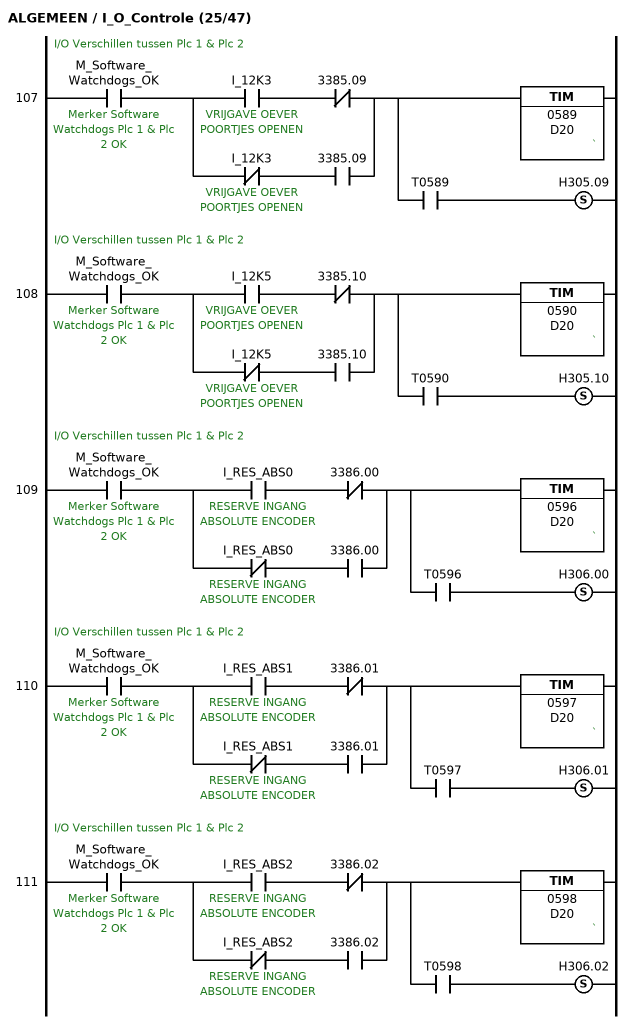
; rung 107: I/O Verschillen tussen Plc 1 & Plc 2
LD M_Software_Watchdogs_OK  ; Merker Software Watchdogs Plc 1 & Plc 2 OK
LD I_12K3  ; VRIJGAVE OEVER POORTJES OPENEN
ANDNOT 3385.09
LDNOT I_12K3  ; VRIJGAVE OEVER POORTJES OPENEN
AND 3385.09
ORLD
ANDLD
TIM 0589 D20  ; `
AND T0589
SET H305.09
; rung 108: I/O Verschillen tussen Plc 1 & Plc 2
LD M_Software_Watchdogs_OK  ; Merker Software Watchdogs Plc 1 & Plc 2 OK
LD I_12K5  ; VRIJGAVE OEVER POORTJES OPENEN
ANDNOT 3385.10
LDNOT I_12K5  ; VRIJGAVE OEVER POORTJES OPENEN
AND 3385.10
ORLD
ANDLD
TIM 0590 D20  ; `
AND T0590
SET H305.10
; rung 109: I/O Verschillen tussen Plc 1 & Plc 2
LD M_Software_Watchdogs_OK  ; Merker Software Watchdogs Plc 1 & Plc 2 OK
LD I_RES_ABS0  ; RESERVE INGANG ABSOLUTE ENCODER
ANDNOT 3386.00
LDNOT I_RES_ABS0  ; RESERVE INGANG ABSOLUTE ENCODER
AND 3386.00
ORLD
ANDLD
TIM 0596 D20  ; `
AND T0596
SET H306.00
; rung 110: I/O Verschillen tussen Plc 1 & Plc 2
LD M_Software_Watchdogs_OK  ; Merker Software Watchdogs Plc 1 & Plc 2 OK
LD I_RES_ABS1  ; RESERVE INGANG ABSOLUTE ENCODER
ANDNOT 3386.01
LDNOT I_RES_ABS1  ; RESERVE INGANG ABSOLUTE ENCODER
AND 3386.01
ORLD
ANDLD
TIM 0597 D20  ; `
AND T0597
SET H306.01
; rung 111: I/O Verschillen tussen Plc 1 & Plc 2
LD M_Software_Watchdogs_OK  ; Merker Software Watchdogs Plc 1 & Plc 2 OK
LD I_RES_ABS2  ; RESERVE INGANG ABSOLUTE ENCODER
ANDNOT 3386.02
LDNOT I_RES_ABS2  ; RESERVE INGANG ABSOLUTE ENCODER
AND 3386.02
ORLD
ANDLD
TIM 0598 D20  ; `
AND T0598
SET H306.02

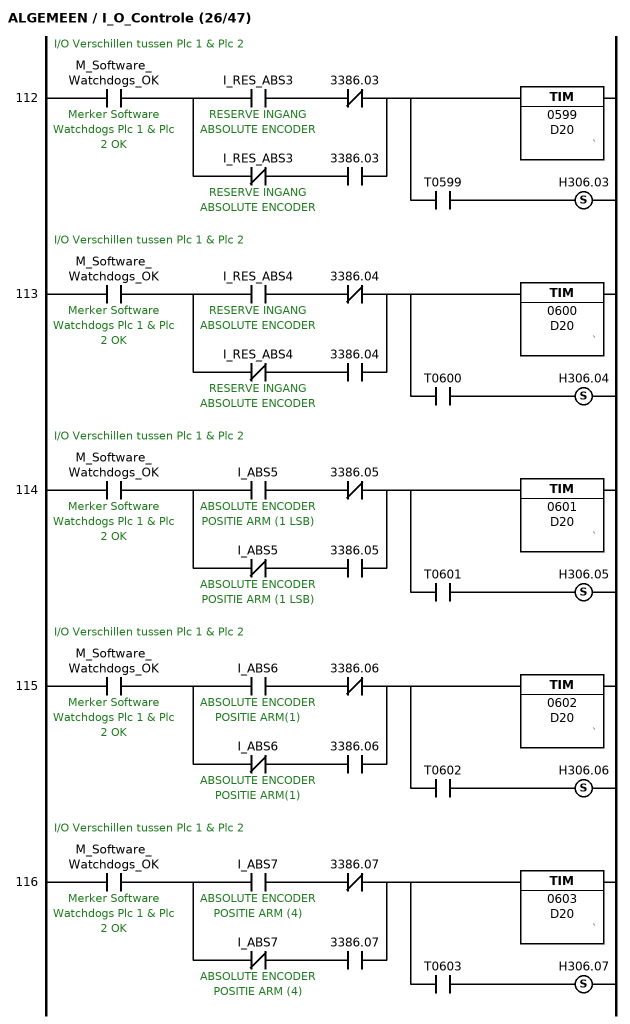
; rung 112: I/O Verschillen tussen Plc 1 & Plc 2
LD M_Software_Watchdogs_OK  ; Merker Software Watchdogs Plc 1 & Plc 2 OK
LD I_RES_ABS3  ; RESERVE INGANG ABSOLUTE ENCODER
ANDNOT 3386.03
LDNOT I_RES_ABS3  ; RESERVE INGANG ABSOLUTE ENCODER
AND 3386.03
ORLD
ANDLD
TIM 0599 D20  ; `
AND T0599
SET H306.03
; rung 113: I/O Verschillen tussen Plc 1 & Plc 2
LD M_Software_Watchdogs_OK  ; Merker Software Watchdogs Plc 1 & Plc 2 OK
LD I_RES_ABS4  ; RESERVE INGANG ABSOLUTE ENCODER
ANDNOT 3386.04
LDNOT I_RES_ABS4  ; RESERVE INGANG ABSOLUTE ENCODER
AND 3386.04
ORLD
ANDLD
TIM 0600 D20  ; `
AND T0600
SET H306.04
; rung 114: I/O Verschillen tussen Plc 1 & Plc 2
LD M_Software_Watchdogs_OK  ; Merker Software Watchdogs Plc 1 & Plc 2 OK
LD I_ABS5  ; ABSOLUTE ENCODER POSITIE ARM (1 LSB)
ANDNOT 3386.05
LDNOT I_ABS5  ; ABSOLUTE ENCODER POSITIE ARM (1 LSB)
AND 3386.05
ORLD
ANDLD
TIM 0601 D20  ; `
AND T0601
SET H306.05
; rung 115: I/O Verschillen tussen Plc 1 & Plc 2
LD M_Software_Watchdogs_OK  ; Merker Software Watchdogs Plc 1 & Plc 2 OK
LD I_ABS6  ; ABSOLUTE ENCODER POSITIE ARM(1)
ANDNOT 3386.06
LDNOT I_ABS6  ; ABSOLUTE ENCODER POSITIE ARM(1)
AND 3386.06
ORLD
ANDLD
TIM 0602 D20  ; `
AND T0602
SET H306.06
; rung 116: I/O Verschillen tussen Plc 1 & Plc 2
LD M_Software_Watchdogs_OK  ; Merker Software Watchdogs Plc 1 & Plc 2 OK
LD I_ABS7  ; ABSOLUTE ENCODER POSITIE ARM (4)
ANDNOT 3386.07
LDNOT I_ABS7  ; ABSOLUTE ENCODER POSITIE ARM (4)
AND 3386.07
ORLD
ANDLD
TIM 0603 D20  ; `
AND T0603
SET H306.07

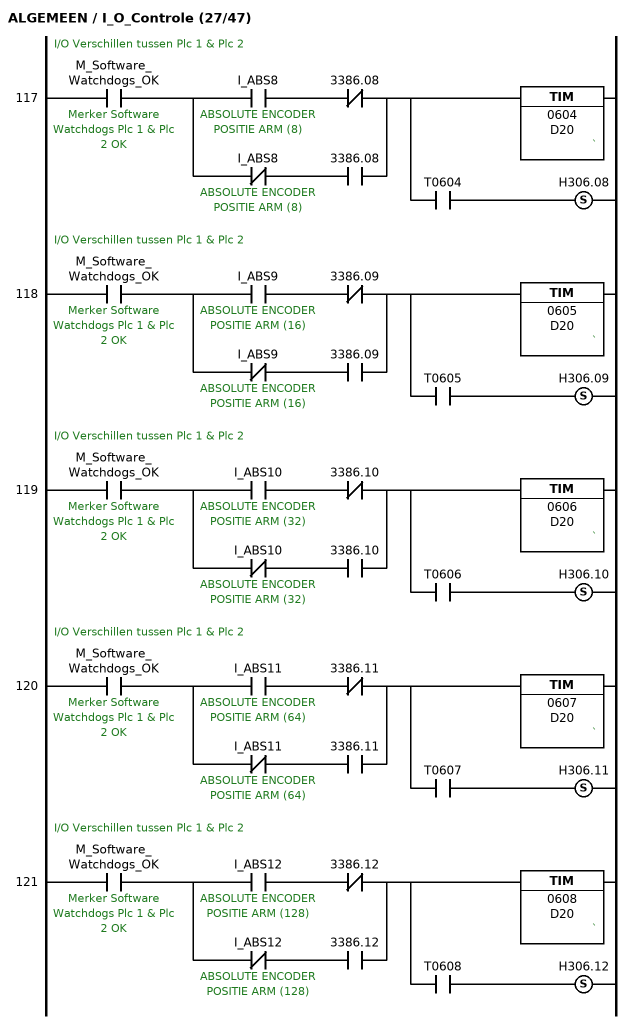
; rung 117: I/O Verschillen tussen Plc 1 & Plc 2
LD M_Software_Watchdogs_OK  ; Merker Software Watchdogs Plc 1 & Plc 2 OK
LD I_ABS8  ; ABSOLUTE ENCODER POSITIE ARM (8)
ANDNOT 3386.08
LDNOT I_ABS8  ; ABSOLUTE ENCODER POSITIE ARM (8)
AND 3386.08
ORLD
ANDLD
TIM 0604 D20  ; `
AND T0604
SET H306.08
; rung 118: I/O Verschillen tussen Plc 1 & Plc 2
LD M_Software_Watchdogs_OK  ; Merker Software Watchdogs Plc 1 & Plc 2 OK
LD I_ABS9  ; ABSOLUTE ENCODER POSITIE ARM (16)
ANDNOT 3386.09
LDNOT I_ABS9  ; ABSOLUTE ENCODER POSITIE ARM (16)
AND 3386.09
ORLD
ANDLD
TIM 0605 D20  ; `
AND T0605
SET H306.09
; rung 119: I/O Verschillen tussen Plc 1 & Plc 2
LD M_Software_Watchdogs_OK  ; Merker Software Watchdogs Plc 1 & Plc 2 OK
LD I_ABS10  ; ABSOLUTE ENCODER POSITIE ARM (32)
ANDNOT 3386.10
LDNOT I_ABS10  ; ABSOLUTE ENCODER POSITIE ARM (32)
AND 3386.10
ORLD
ANDLD
TIM 0606 D20  ; `
AND T0606
SET H306.10
; rung 120: I/O Verschillen tussen Plc 1 & Plc 2
LD M_Software_Watchdogs_OK  ; Merker Software Watchdogs Plc 1 & Plc 2 OK
LD I_ABS11  ; ABSOLUTE ENCODER POSITIE ARM (64)
ANDNOT 3386.11
LDNOT I_ABS11  ; ABSOLUTE ENCODER POSITIE ARM (64)
AND 3386.11
ORLD
ANDLD
TIM 0607 D20  ; `
AND T0607
SET H306.11
; rung 121: I/O Verschillen tussen Plc 1 & Plc 2
LD M_Software_Watchdogs_OK  ; Merker Software Watchdogs Plc 1 & Plc 2 OK
LD I_ABS12  ; ABSOLUTE ENCODER POSITIE ARM (128)
ANDNOT 3386.12
LDNOT I_ABS12  ; ABSOLUTE ENCODER POSITIE ARM (128)
AND 3386.12
ORLD
ANDLD
TIM 0608 D20  ; `
AND T0608
SET H306.12

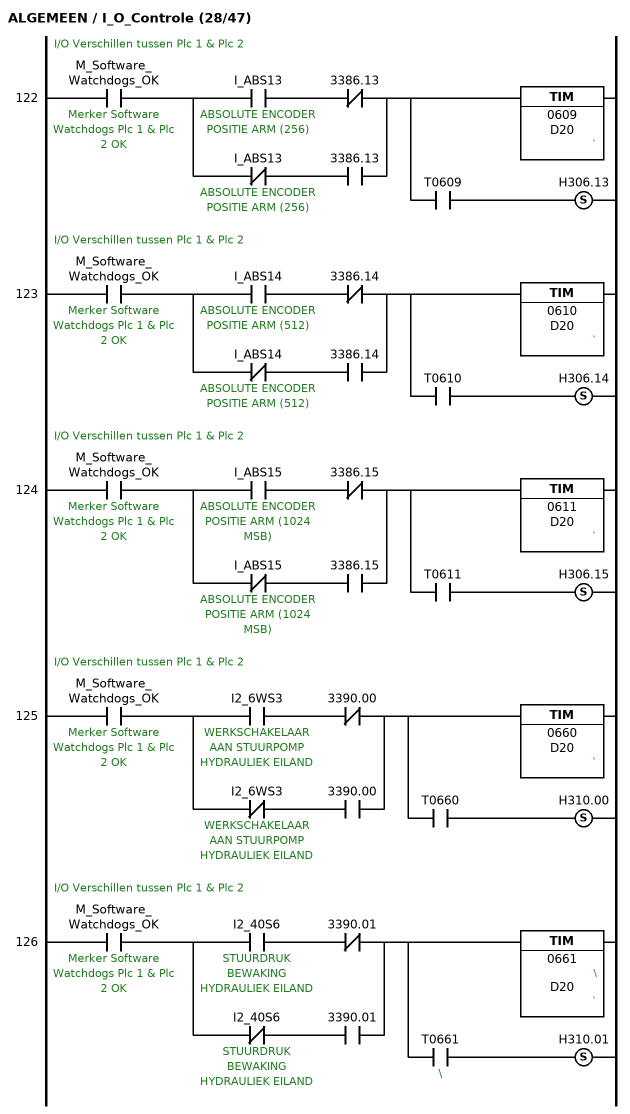
; rung 122: I/O Verschillen tussen Plc 1 & Plc 2
LD M_Software_Watchdogs_OK  ; Merker Software Watchdogs Plc 1 & Plc 2 OK
LD I_ABS13  ; ABSOLUTE ENCODER POSITIE ARM (256)
ANDNOT 3386.13
LDNOT I_ABS13  ; ABSOLUTE ENCODER POSITIE ARM (256)
AND 3386.13
ORLD
ANDLD
TIM 0609 D20  ; `
AND T0609
SET H306.13
; rung 123: I/O Verschillen tussen Plc 1 & Plc 2
LD M_Software_Watchdogs_OK  ; Merker Software Watchdogs Plc 1 & Plc 2 OK
LD I_ABS14  ; ABSOLUTE ENCODER POSITIE ARM (512)
ANDNOT 3386.14
LDNOT I_ABS14  ; ABSOLUTE ENCODER POSITIE ARM (512)
AND 3386.14
ORLD
ANDLD
TIM 0610 D20  ; `
AND T0610
SET H306.14
; rung 124: I/O Verschillen tussen Plc 1 & Plc 2
LD M_Software_Watchdogs_OK  ; Merker Software Watchdogs Plc 1 & Plc 2 OK
LD I_ABS15  ; ABSOLUTE ENCODER POSITIE ARM (1024 MSB)
ANDNOT 3386.15
LDNOT I_ABS15  ; ABSOLUTE ENCODER POSITIE ARM (1024 MSB)
AND 3386.15
ORLD
ANDLD
TIM 0611 D20  ; `
AND T0611
SET H306.15
; rung 125: I/O Verschillen tussen Plc 1 & Plc 2
LD M_Software_Watchdogs_OK  ; Merker Software Watchdogs Plc 1 & Plc 2 OK
LD I2_6WS3  ; WERKSCHAKELAAR AAN STUURPOMP HYDRAULIEK EILAND
ANDNOT 3390.00
LDNOT I2_6WS3  ; WERKSCHAKELAAR AAN STUURPOMP HYDRAULIEK EILAND
AND 3390.00
ORLD
ANDLD
TIM 0660 D20  ; `
AND T0660
SET H310.00
; rung 126: I/O Verschillen tussen Plc 1 & Plc 2
LD M_Software_Watchdogs_OK  ; Merker Software Watchdogs Plc 1 & Plc 2 OK
LD I2_40S6  ; STUURDRUK BEWAKING HYDRAULIEK EILAND
ANDNOT 3390.01
LDNOT I2_40S6  ; STUURDRUK BEWAKING HYDRAULIEK EILAND
AND 3390.01
ORLD
ANDLD
TIM 0661 D20  ; `, \
AND T0661  ; \
SET H310.01

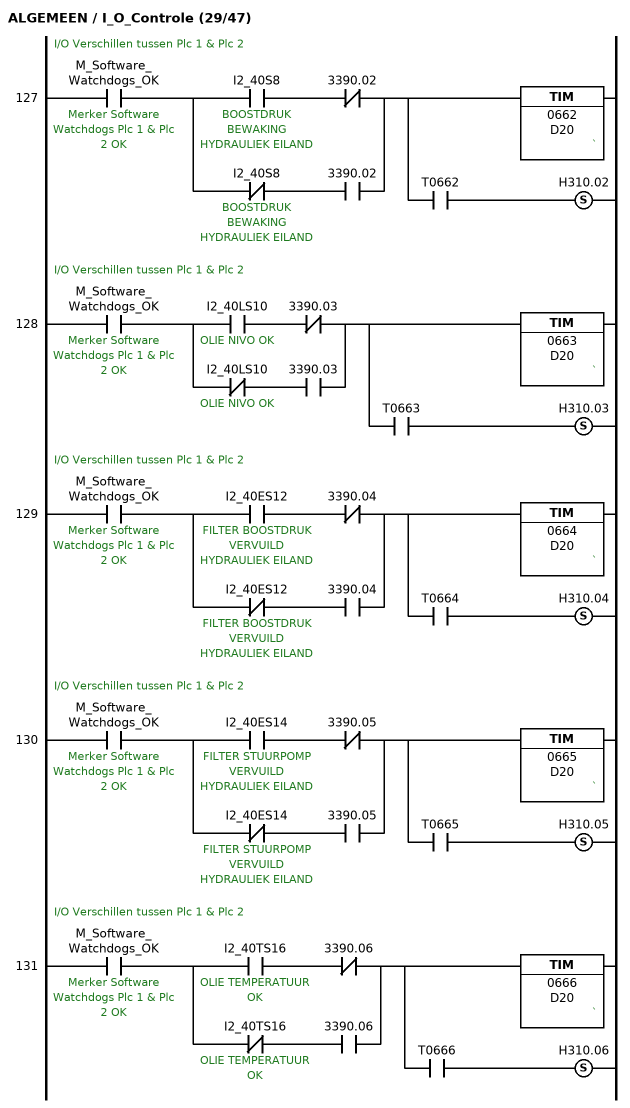
; rung 127: I/O Verschillen tussen Plc 1 & Plc 2
LD M_Software_Watchdogs_OK  ; Merker Software Watchdogs Plc 1 & Plc 2 OK
LD I2_40S8  ; BOOSTDRUK BEWAKING HYDRAULIEK EILAND
ANDNOT 3390.02
LDNOT I2_40S8  ; BOOSTDRUK BEWAKING HYDRAULIEK EILAND
AND 3390.02
ORLD
ANDLD
TIM 0662 D20  ; `
AND T0662
SET H310.02
; rung 128: I/O Verschillen tussen Plc 1 & Plc 2
LD M_Software_Watchdogs_OK  ; Merker Software Watchdogs Plc 1 & Plc 2 OK
LD I2_40LS10  ; OLIE NIVO OK
ANDNOT 3390.03
LDNOT I2_40LS10  ; OLIE NIVO OK
AND 3390.03
ORLD
ANDLD
TIM 0663 D20  ; `
AND T0663
SET H310.03
; rung 129: I/O Verschillen tussen Plc 1 & Plc 2
LD M_Software_Watchdogs_OK  ; Merker Software Watchdogs Plc 1 & Plc 2 OK
LD I2_40ES12  ; FILTER BOOSTDRUK VERVUILD HYDRAULIEK EILAND
ANDNOT 3390.04
LDNOT I2_40ES12  ; FILTER BOOSTDRUK VERVUILD HYDRAULIEK EILAND
AND 3390.04
ORLD
ANDLD
TIM 0664 D20  ; `
AND T0664
SET H310.04
; rung 130: I/O Verschillen tussen Plc 1 & Plc 2
LD M_Software_Watchdogs_OK  ; Merker Software Watchdogs Plc 1 & Plc 2 OK
LD I2_40ES14  ; FILTER STUURPOMP VERVUILD HYDRAULIEK EILAND
ANDNOT 3390.05
LDNOT I2_40ES14  ; FILTER STUURPOMP VERVUILD HYDRAULIEK EILAND
AND 3390.05
ORLD
ANDLD
TIM 0665 D20  ; `
AND T0665
SET H310.05
; rung 131: I/O Verschillen tussen Plc 1 & Plc 2
LD M_Software_Watchdogs_OK  ; Merker Software Watchdogs Plc 1 & Plc 2 OK
LD I2_40TS16  ; OLIE TEMPERATUUR OK
ANDNOT 3390.06
LDNOT I2_40TS16  ; OLIE TEMPERATUUR OK
AND 3390.06
ORLD
ANDLD
TIM 0666 D20  ; `
AND T0666
SET H310.06

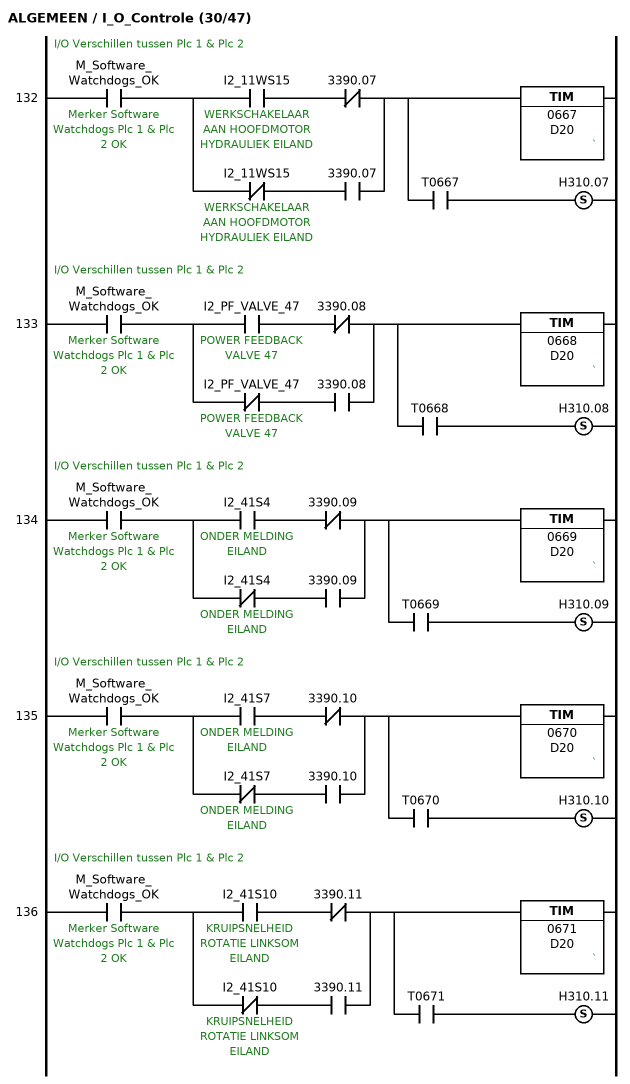
; rung 132: I/O Verschillen tussen Plc 1 & Plc 2
LD M_Software_Watchdogs_OK  ; Merker Software Watchdogs Plc 1 & Plc 2 OK
LD I2_11WS15  ; WERKSCHAKELAAR AAN HOOFDMOTOR HYDRAULIEK EILAND
ANDNOT 3390.07
LDNOT I2_11WS15  ; WERKSCHAKELAAR AAN HOOFDMOTOR HYDRAULIEK EILAND
AND 3390.07
ORLD
ANDLD
TIM 0667 D20  ; `
AND T0667
SET H310.07
; rung 133: I/O Verschillen tussen Plc 1 & Plc 2
LD M_Software_Watchdogs_OK  ; Merker Software Watchdogs Plc 1 & Plc 2 OK
LD I2_PF_VALVE_47  ; POWER FEEDBACK VALVE 47
ANDNOT 3390.08
LDNOT I2_PF_VALVE_47  ; POWER FEEDBACK VALVE 47
AND 3390.08
ORLD
ANDLD
TIM 0668 D20  ; `
AND T0668
SET H310.08
; rung 134: I/O Verschillen tussen Plc 1 & Plc 2
LD M_Software_Watchdogs_OK  ; Merker Software Watchdogs Plc 1 & Plc 2 OK
LD I2_41S4  ; ONDER MELDING EILAND
ANDNOT 3390.09
LDNOT I2_41S4  ; ONDER MELDING EILAND
AND 3390.09
ORLD
ANDLD
TIM 0669 D20  ; `
AND T0669
SET H310.09
; rung 135: I/O Verschillen tussen Plc 1 & Plc 2
LD M_Software_Watchdogs_OK  ; Merker Software Watchdogs Plc 1 & Plc 2 OK
LD I2_41S7  ; ONDER MELDING EILAND
ANDNOT 3390.10
LDNOT I2_41S7  ; ONDER MELDING EILAND
AND 3390.10
ORLD
ANDLD
TIM 0670 D20  ; `
AND T0670
SET H310.10
; rung 136: I/O Verschillen tussen Plc 1 & Plc 2
LD M_Software_Watchdogs_OK  ; Merker Software Watchdogs Plc 1 & Plc 2 OK
LD I2_41S10  ; KRUIPSNELHEID ROTATIE LINKSOM EILAND
ANDNOT 3390.11
LDNOT I2_41S10  ; KRUIPSNELHEID ROTATIE LINKSOM EILAND
AND 3390.11
ORLD
ANDLD
TIM 0671 D20  ; `
AND T0671
SET H310.11

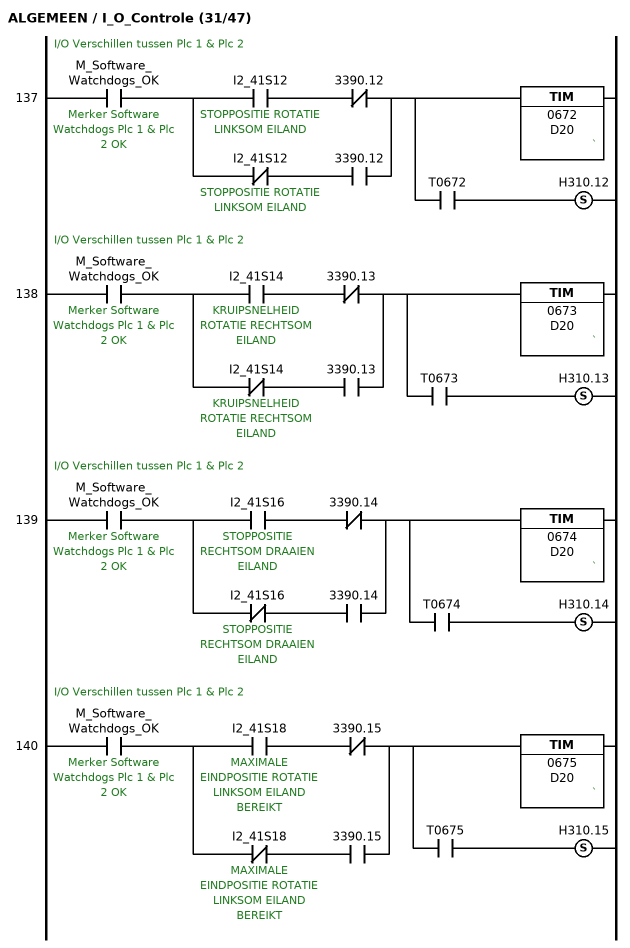
; rung 137: I/O Verschillen tussen Plc 1 & Plc 2
LD M_Software_Watchdogs_OK  ; Merker Software Watchdogs Plc 1 & Plc 2 OK
LD I2_41S12  ; STOPPOSITIE ROTATIE LINKSOM EILAND
ANDNOT 3390.12
LDNOT I2_41S12  ; STOPPOSITIE ROTATIE LINKSOM EILAND
AND 3390.12
ORLD
ANDLD
TIM 0672 D20  ; `
AND T0672
SET H310.12
; rung 138: I/O Verschillen tussen Plc 1 & Plc 2
LD M_Software_Watchdogs_OK  ; Merker Software Watchdogs Plc 1 & Plc 2 OK
LD I2_41S14  ; KRUIPSNELHEID ROTATIE RECHTSOM EILAND
ANDNOT 3390.13
LDNOT I2_41S14  ; KRUIPSNELHEID ROTATIE RECHTSOM EILAND
AND 3390.13
ORLD
ANDLD
TIM 0673 D20  ; `
AND T0673
SET H310.13
; rung 139: I/O Verschillen tussen Plc 1 & Plc 2
LD M_Software_Watchdogs_OK  ; Merker Software Watchdogs Plc 1 & Plc 2 OK
LD I2_41S16  ; STOPPOSITIE RECHTSOM DRAAIEN EILAND
ANDNOT 3390.14
LDNOT I2_41S16  ; STOPPOSITIE RECHTSOM DRAAIEN EILAND
AND 3390.14
ORLD
ANDLD
TIM 0674 D20  ; `
AND T0674
SET H310.14
; rung 140: I/O Verschillen tussen Plc 1 & Plc 2
LD M_Software_Watchdogs_OK  ; Merker Software Watchdogs Plc 1 & Plc 2 OK
LD I2_41S18  ; MAXIMALE EINDPOSITIE ROTATIE LINKSOM EILAND BEREIKT
ANDNOT 3390.15
LDNOT I2_41S18  ; MAXIMALE EINDPOSITIE ROTATIE LINKSOM EILAND BEREIKT
AND 3390.15
ORLD
ANDLD
TIM 0675 D20  ; `
AND T0675
SET H310.15

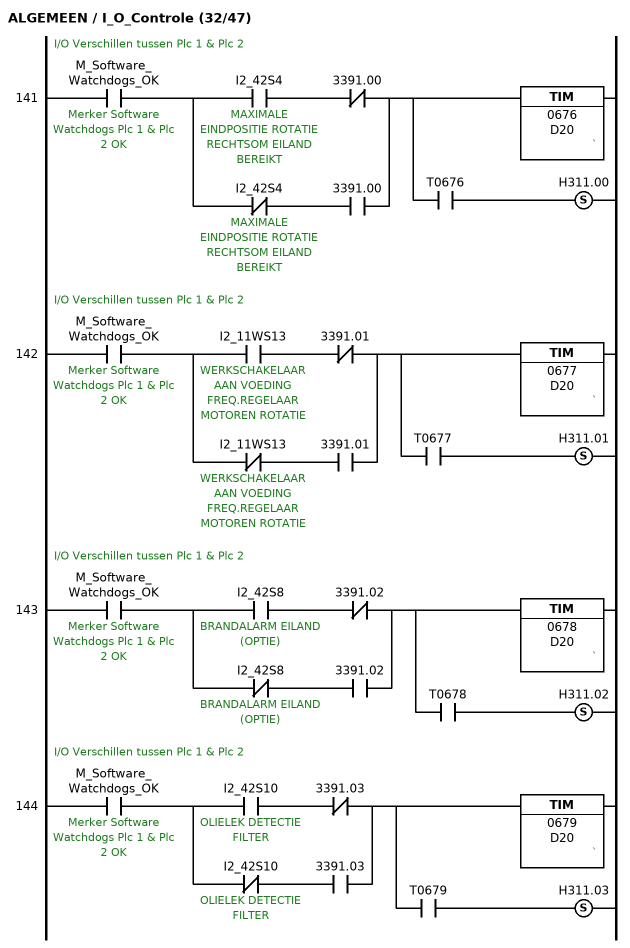
; rung 141: I/O Verschillen tussen Plc 1 & Plc 2
LD M_Software_Watchdogs_OK  ; Merker Software Watchdogs Plc 1 & Plc 2 OK
LD I2_42S4  ; MAXIMALE EINDPOSITIE ROTATIE RECHTSOM EILAND BEREIKT
ANDNOT 3391.00
LDNOT I2_42S4  ; MAXIMALE EINDPOSITIE ROTATIE RECHTSOM EILAND BEREIKT
AND 3391.00
ORLD
ANDLD
TIM 0676 D20  ; `
AND T0676
SET H311.00
; rung 142: I/O Verschillen tussen Plc 1 & Plc 2
LD M_Software_Watchdogs_OK  ; Merker Software Watchdogs Plc 1 & Plc 2 OK
LD I2_11WS13  ; WERKSCHAKELAAR AAN VOEDING FREQ.REGELAAR MOTOREN ROTATIE
ANDNOT 3391.01
LDNOT I2_11WS13  ; WERKSCHAKELAAR AAN VOEDING FREQ.REGELAAR MOTOREN ROTATIE
AND 3391.01
ORLD
ANDLD
TIM 0677 D20  ; `
AND T0677
SET H311.01
; rung 143: I/O Verschillen tussen Plc 1 & Plc 2
LD M_Software_Watchdogs_OK  ; Merker Software Watchdogs Plc 1 & Plc 2 OK
LD I2_42S8  ; BRANDALARM EILAND (OPTIE)
ANDNOT 3391.02
LDNOT I2_42S8  ; BRANDALARM EILAND (OPTIE)
AND 3391.02
ORLD
ANDLD
TIM 0678 D20  ; `
AND T0678
SET H311.02
; rung 144: I/O Verschillen tussen Plc 1 & Plc 2
LD M_Software_Watchdogs_OK  ; Merker Software Watchdogs Plc 1 & Plc 2 OK
LD I2_42S10  ; OLIELEK DETECTIE FILTER
ANDNOT 3391.03
LDNOT I2_42S10  ; OLIELEK DETECTIE FILTER
AND 3391.03
ORLD
ANDLD
TIM 0679 D20  ; `
AND T0679
SET H311.03

